  MoveL 3991 to (-40.74, 149.76, 69.25) mm, rotated rx -180 ry 0 rz 180 deg; joints [-126.379, -59.707, -80.826, 60.372, 67.852, -33.54]
  MoveL 3992 to (-40.74, 149.76, 69.25) mm, rotated rx -180 ry 0 rz 180 deg; joints [-126.379, -59.707, -80.826, 60.372, 67.852, -33.54]
  Call Extruder(12.04180)
  MoveL 3993 to (-40.78, 149.45, 69.25) mm, rotated rx 180 ry 0 rz 180 deg; joints [-126.398, -59.688, -80.879, 60.344, 67.858, -33.503]
  MoveL 3994 to (-40.78, 149.45, 69.25) mm, rotated rx 180 ry 0 rz 180 deg; joints [-126.398, -59.688, -80.879, 60.344, 67.858, -33.503]
  Call Extruder(12.20062)
  MoveL 3995 to (-40.83, 149.14, 69.25) mm, rotated rx 180 ry 0 rz -180 deg; joints [-126.417, -59.668, -80.931, 60.315, 67.863, -33.466]
  MoveL 3996 to (-40.83, 149.14, 69.25) mm, rotated rx 180 ry 0 rz -180 deg; joints [-126.417, -59.668, -80.931, 60.315, 67.863, -33.466]
  Call Extruder(12.37928)
  MoveL 3997 to (-40.88, 148.8, 69.25) mm, rotated rx 180 ry 0 rz 180 deg; joints [-126.439, -59.646, -80.989, 60.282, 67.869, -33.424]
  MoveL 3998 to (-40.88, 148.8, 69.25) mm, rotated rx 180 ry 0 rz 180 deg; joints [-126.439, -59.646, -80.989, 60.282, 67.869, -33.424]
  Call Extruder(12.57772)
  MoveL 3999 to (-40.92, 148.41, 69.25) mm, rotated rx 180 ry 0 rz 180 deg; joints [-126.465, -59.622, -81.054, 60.244, 67.875, -33.377]
  MoveL 4000 to (-40.92, 148.41, 69.25) mm, rotated rx 180 ry 0 rz 180 deg; joints [-126.465, -59.622, -81.054, 60.244, 67.875, -33.377]
  Call Extruder(12.77530)
  MoveL 4001 to (-40.97, 148.02, 69.25) mm, rotated rx 180 ry 0 rz 180 deg; joints [-126.491, -59.598, -81.118, 60.206, 67.881, -33.33]
  MoveL 4002 to (-40.97, 148.02, 69.25) mm, rotated rx 180 ry 0 rz 180 deg; joints [-126.491, -59.598, -81.118, 60.206, 67.881, -33.33]
  Call Extruder(12.97200)
  MoveL 4003 to (-41.02, 147.63, 69.25) mm, rotated rx 180 ry 0 rz 180 deg; joints [-126.517, -59.574, -81.183, 60.168, 67.886, -33.284]
  MoveL 4004 to (-41.02, 147.63, 69.25) mm, rotated rx 180 ry 0 rz 180 deg; joints [-126.517, -59.574, -81.183, 60.168, 67.886, -33.284]
  Call Extruder(13.16784)
  MoveL 4005 to (-41.06, 147.25, 69.25) mm, rotated rx 180 ry 0 rz 180 deg; joints [-126.543, -59.55, -81.247, 60.131, 67.892, -33.237]
  MoveL 4006 to (-41.06, 147.25, 69.25) mm, rotated rx 180 ry 0 rz 180 deg; joints [-126.543, -59.55, -81.247, 60.131, 67.892, -33.237]
  Call Extruder(13.46324)
  MoveL 4007 to (-41.11, 146.66, 69.25) mm, rotated rx 180 ry 0 rz 180 deg; joints [-126.585, -59.515, -81.342, 60.071, 67.899, -33.167]
  MoveL 4008 to (-41.11, 146.66, 69.25) mm, rotated rx 180 ry 0 rz 180 deg; joints [-126.585, -59.515, -81.342, 60.071, 67.899, -33.167]
  Call Extruder(13.75731)
  MoveL 4009 to (-41.15, 146.07, 69.25) mm, rotated rx -180 ry 0 rz 180 deg; joints [-126.628, -59.48, -81.437, 60.012, 67.906, -33.096]
  MoveL 4010 to (-41.15, 146.07, 69.25) mm, rotated rx -180 ry 0 rz 180 deg; joints [-126.628, -59.48, -81.437, 60.012, 67.906, -33.096]
  Call Extruder(14.05004)
  MoveL 4011 to (-41.2, 145.48, 69.25) mm, rotated rx -180 ry 0 rz -180 deg; joints [-126.67, -59.444, -81.532, 59.953, 67.912, -33.026]
  MoveL 4012 to (-41.2, 145.48, 69.25) mm, rotated rx -180 ry 0 rz -180 deg; joints [-126.67, -59.444, -81.532, 59.953, 67.912, -33.026]
  Call Extruder(14.62350)
  MoveL 4013 to (-41.25, 144.32, 69.25) mm, rotated rx 180 ry 0 rz -180 deg; joints [-126.759, -59.377, -81.714, 59.832, 67.921, -32.889]
  MoveL 4014 to (-41.25, 144.32, 69.25) mm, rotated rx 180 ry 0 rz -180 deg; joints [-126.759, -59.377, -81.714, 59.832, 67.921, -32.889]
  Call Extruder(15.33745)
  MoveL 4015 to (-41.29, 142.86, 69.25) mm, rotated rx 180 ry 0 rz 180 deg; joints [-126.873, -59.294, -81.938, 59.679, 67.931, -32.718]
  Call Extruder(57.40228)
  MoveL 4016 to (-41.29, 57.14, 69.25) mm, rotated rx 180 ry 0 rz 180 deg; joints [-135.148, -55.35, -93.55, 49.281, 68.519, -23.047]
  Call Extruder(57.83083)
  MoveL 4017 to (-41.27, 56.26, 69.25) mm, rotated rx -180 ry 0 rz 180 deg; joints [-135.25, -55.319, -93.653, 49.16, 68.526, -22.952]
  MoveL 4018 to (-41.27, 56.26, 69.25) mm, rotated rx -180 ry 0 rz 180 deg; joints [-135.25, -55.319, -93.653, 49.16, 68.526, -22.952]
  Call Extruder(58.40429)
  MoveL 4019 to (-41.23, 55.1, 69.25) mm, rotated rx -180 ry 0 rz -180 deg; joints [-135.387, -55.278, -93.786, 48.995, 68.534, -22.827]
  MoveL 4020 to (-41.23, 55.1, 69.25) mm, rotated rx -180 ry 0 rz -180 deg; joints [-135.387, -55.278, -93.786, 48.995, 68.534, -22.827]
  Call Extruder(58.83860)
  MoveL 4021 to (-41.18, 54.23, 69.25) mm, rotated rx 180 ry 0 rz 180 deg; joints [-135.493, -55.248, -93.885, 48.87, 68.538, -22.733]
  MoveL 4022 to (-41.18, 54.23, 69.25) mm, rotated rx 180 ry 0 rz 180 deg; joints [-135.493, -55.248, -93.885, 48.87, 68.538, -22.733]
  Call Extruder(59.13267)
  MoveL 4023 to (-41.13, 53.64, 69.25) mm, rotated rx -180 ry 0 rz 180 deg; joints [-135.566, -55.228, -93.95, 48.784, 68.539, -22.67]
  MoveL 4024 to (-41.13, 53.64, 69.25) mm, rotated rx -180 ry 0 rz 180 deg; joints [-135.566, -55.228, -93.95, 48.784, 68.539, -22.67]
  Call Extruder(59.42806)
  MoveL 4025 to (-41.09, 53.05, 69.25) mm, rotated rx -180 ry 0 rz 180 deg; joints [-135.64, -55.209, -94.014, 48.699, 68.541, -22.607]
  MoveL 4026 to (-41.09, 53.05, 69.25) mm, rotated rx -180 ry 0 rz 180 deg; joints [-135.64, -55.209, -94.014, 48.699, 68.541, -22.607]
  Call Extruder(59.67430)
  MoveL 4027 to (-41.04, 52.56, 69.25) mm, rotated rx 180 ry 0 rz -180 deg; joints [-135.701, -55.193, -94.066, 48.627, 68.541, -22.556]
  MoveL 4028 to (-41.04, 52.56, 69.25) mm, rotated rx 180 ry 0 rz -180 deg; joints [-135.701, -55.193, -94.066, 48.627, 68.541, -22.556]
  Call Extruder(59.87100)
  MoveL 4029 to (-40.99, 52.17, 69.25) mm, rotated rx -180 ry 0 rz 180 deg; joints [-135.751, -55.181, -94.107, 48.569, 68.54, -22.515]
  MoveL 4030 to (-40.99, 52.17, 69.25) mm, rotated rx -180 ry 0 rz 180 deg; joints [-135.751, -55.181, -94.107, 48.569, 68.54, -22.515]
  Call Extruder(60.06858)
  MoveL 4031 to (-40.95, 51.78, 69.25) mm, rotated rx 180 ry 0 rz -180 deg; joints [-135.801, -55.169, -94.147, 48.511, 68.54, -22.474]
  MoveL 4032 to (-40.95, 51.78, 69.25) mm, rotated rx 180 ry 0 rz -180 deg; joints [-135.801, -55.169, -94.147, 48.511, 68.54, -22.474]
  Call Extruder(60.26702)
  MoveL 4033 to (-40.9, 51.4, 69.25) mm, rotated rx 180 ry 0 rz -180 deg; joints [-135.852, -55.157, -94.187, 48.453, 68.539, -22.433]
  MoveL 4034 to (-40.9, 51.4, 69.25) mm, rotated rx 180 ry 0 rz -180 deg; joints [-135.852, -55.157, -94.187, 48.453, 68.539, -22.433]
  Call Extruder(60.46633)
  MoveL 4035 to (-40.86, 51.01, 69.25) mm, rotated rx 180 ry 0 rz 180 deg; joints [-135.902, -55.145, -94.227, 48.394, 68.539, -22.392]
  MoveL 4036 to (-40.86, 51.01, 69.25) mm, rotated rx 180 ry 0 rz 180 deg; joints [-135.902, -55.145, -94.227, 48.394, 68.539, -22.392]
  Call Extruder(60.62514)
  MoveL 4037 to (-40.81, 50.7, 69.25) mm, rotated rx 180 ry 0 rz -180 deg; joints [-135.943, -55.136, -94.257, 48.347, 68.537, -22.36]
  MoveL 4038 to (-40.81, 50.7, 69.25) mm, rotated rx 180 ry 0 rz -180 deg; joints [-135.943, -55.136, -94.257, 48.347, 68.537, -22.36]
  Call Extruder(60.78469)
  MoveL 4039 to (-40.76, 50.4, 69.25) mm, rotated rx 180 ry 0 rz -180 deg; joints [-135.984, -55.127, -94.287, 48.3, 68.535, -22.329]
  MoveL 4040 to (-40.76, 50.4, 69.25) mm, rotated rx 180 ry 0 rz -180 deg; joints [-135.984, -55.127, -94.287, 48.3, 68.535, -22.329]
  Call Extruder(60.94496)
  MoveL 4041 to (-40.71, 50.09, 69.25) mm, rotated rx 180 ry 0 rz 180 deg; joints [-136.025, -55.118, -94.317, 48.253, 68.534, -22.297]
  MoveL 4042 to (-40.71, 50.09, 69.25) mm, rotated rx 180 ry 0 rz 180 deg; joints [-136.025, -55.118, -94.317, 48.253, 68.534, -22.297]
  Call Extruder(61.10596)
  MoveL 4043 to (-40.66, 49.79, 69.25) mm, rotated rx 180 ry 0 rz -180 deg; joints [-136.067, -55.109, -94.347, 48.206, 68.532, -22.265]
  MoveL 4044 to (-40.66, 49.79, 69.25) mm, rotated rx 180 ry 0 rz -180 deg; joints [-136.067, -55.109, -94.347, 48.206, 68.532, -22.265]
  Call Extruder(61.26769)
  MoveL 4045 to (-40.61, 49.48, 69.25) mm, rotated rx 180 ry 0 rz 180 deg; joints [-136.108, -55.1, -94.377, 48.159, 68.53, -22.233]
  MoveL 4046 to (-40.61, 49.48, 69.25) mm, rotated rx 180 ry 0 rz 180 deg; joints [-136.108, -55.1, -94.377, 48.159, 68.53, -22.233]
  Call Extruder(61.43014)
  MoveL 4047 to (-40.56, 49.18, 69.25) mm, rotated rx 180 ry 0 rz 180 deg; joints [-136.149, -55.091, -94.407, 48.112, 68.529, -22.201]
  MoveL 4048 to (-40.56, 49.18, 69.25) mm, rotated rx 180 ry 0 rz 180 deg; joints [-136.149, -55.091, -94.407, 48.112, 68.529, -22.201]
  Call Extruder(61.56407)
  MoveL 4049 to (-40.52, 48.93, 69.25) mm, rotated rx 180 ry 0 rz 180 deg; joints [-136.184, -55.084, -94.43, 48.072, 68.526, -22.176]
  MoveL 4050 to (-40.52, 48.93, 69.25) mm, rotated rx 180 ry 0 rz 180 deg; joints [-136.184, -55.084, -94.43, 48.072, 68.526, -22.176]
  Call Extruder(61.69860)
  MoveL 4051 to (-40.47, 48.68, 69.25) mm, rotated rx 180 ry 0 rz 180 deg; joints [-136.219, -55.077, -94.453, 48.033, 68.524, -22.15]
  MoveL 4052 to (-40.47, 48.68, 69.25) mm, rotated rx 180 ry 0 rz 180 deg; joints [-136.219, -55.077, -94.453, 48.033, 68.524, -22.15]
  Call Extruder(61.83375)
  MoveL 4053 to (-40.42, 48.43, 69.25) mm, rotated rx -180 ry 0 rz -180 deg; joints [-136.254, -55.07, -94.476, 47.993, 68.522, -22.124]
  MoveL 4054 to (-40.42, 48.43, 69.25) mm, rotated rx -180 ry 0 rz -180 deg; joints [-136.254, -55.07, -94.476, 47.993, 68.522, -22.124]
  Call Extruder(61.96950)
  MoveL 4055 to (-40.37, 48.18, 69.25) mm, rotated rx -180 ry 0 rz 180 deg; joints [-136.288, -55.063, -94.499, 47.954, 68.519, -22.099]
  MoveL 4056 to (-40.37, 48.18, 69.25) mm, rotated rx -180 ry 0 rz 180 deg; joints [-136.288, -55.063, -94.499, 47.954, 68.519, -22.099]
  Call Extruder(62.10587)
  MoveL 4057 to (-40.32, 47.93, 69.25) mm, rotated rx 180 ry 0 rz 180 deg; joints [-136.323, -55.056, -94.522, 47.915, 68.517, -22.073]
  MoveL 4058 to (-40.32, 47.93, 69.25) mm, rotated rx 180 ry 0 rz 180 deg; joints [-136.323, -55.056, -94.522, 47.915, 68.517, -22.073]
  Call Extruder(62.24285)
  MoveL 4059 to (-40.27, 47.68, 69.25) mm, rotated rx -180 ry 0 rz 180 deg; joints [-136.358, -55.049, -94.545, 47.875, 68.515, -22.048]
  MoveL 4060 to (-40.27, 47.68, 69.25) mm, rotated rx -180 ry 0 rz 180 deg; joints [-136.358, -55.049, -94.545, 47.875, 68.515, -22.048]
  Call Extruder(62.38043)
  MoveL 4061 to (-40.22, 47.43, 69.25) mm, rotated rx 180 ry 0 rz 180 deg; joints [-136.393, -55.042, -94.568, 47.836, 68.512, -22.022]
  MoveL 4062 to (-40.22, 47.43, 69.25) mm, rotated rx 180 ry 0 rz 180 deg; joints [-136.393, -55.042, -94.568, 47.836, 68.512, -22.022]
  Call Extruder(62.49416)
  MoveL 4063 to (-40.17, 47.23, 69.25) mm, rotated rx -180 ry 0 rz -180 deg; joints [-136.422, -55.037, -94.587, 47.803, 68.51, -22.001]
  MoveL 4064 to (-40.17, 47.23, 69.25) mm, rotated rx -180 ry 0 rz -180 deg; joints [-136.422, -55.037, -94.587, 47.803, 68.51, -22.001]
  Call Extruder(62.60834)
  MoveL 4065 to (-40.13, 47.02, 69.25) mm, rotated rx 180 ry 0 rz 180 deg; joints [-136.452, -55.032, -94.605, 47.77, 68.508, -21.98]
  MoveL 4066 to (-40.13, 47.02, 69.25) mm, rotated rx 180 ry 0 rz 180 deg; joints [-136.452, -55.032, -94.605, 47.77, 68.508, -21.98]
  Call Extruder(62.72297)
  MoveL 4067 to (-40.08, 46.82, 69.25) mm, rotated rx 180 ry 0 rz 180 deg; joints [-136.481, -55.026, -94.623, 47.737, 68.506, -21.959]
  MoveL 4068 to (-40.08, 46.82, 69.25) mm, rotated rx 180 ry 0 rz 180 deg; joints [-136.481, -55.026, -94.623, 47.737, 68.506, -21.959]
  Call Extruder(62.83806)
  MoveL 4069 to (-40.04, 46.61, 69.25) mm, rotated rx 180 ry 0 rz 180 deg; joints [-136.51, -55.021, -94.641, 47.704, 68.503, -21.939]
  MoveL 4070 to (-40.04, 46.61, 69.25) mm, rotated rx 180 ry 0 rz 180 deg; joints [-136.51, -55.021, -94.641, 47.704, 68.503, -21.939]
  Call Extruder(62.96029)
  MoveL 4071 to (-39.98, 46.4, 69.25) mm, rotated rx 180 ry 0 rz 180 deg; joints [-136.542, -55.015, -94.659, 47.669, 68.5, -21.917]
  MoveL 4072 to (-39.98, 46.4, 69.25) mm, rotated rx 180 ry 0 rz 180 deg; joints [-136.542, -55.015, -94.659, 47.669, 68.5, -21.917]
  Call Extruder(63.08996)
  MoveL 4073 to (-39.92, 46.18, 69.25) mm, rotated rx 180 ry 0 rz -180 deg; joints [-136.576, -55.01, -94.677, 47.631, 68.496, -21.895]
  MoveL 4074 to (-39.92, 46.18, 69.25) mm, rotated rx 180 ry 0 rz -180 deg; joints [-136.576, -55.01, -94.677, 47.631, 68.496, -21.895]
  Call Extruder(63.22019)
  MoveL 4075 to (-39.85, 45.95, 69.25) mm, rotated rx 180 ry 0 rz 180 deg; joints [-136.61, -55.005, -94.695, 47.594, 68.491, -21.872]
  MoveL 4076 to (-39.85, 45.95, 69.25) mm, rotated rx 180 ry 0 rz 180 deg; joints [-136.61, -55.005, -94.695, 47.594, 68.491, -21.872]
  Call Extruder(63.35098)
  MoveL 4077 to (-39.78, 45.73, 69.25) mm, rotated rx 180 ry 0 rz 180 deg; joints [-136.644, -55, -94.712, 47.556, 68.487, -21.85]
  MoveL 4078 to (-39.78, 45.73, 69.25) mm, rotated rx 180 ry 0 rz 180 deg; joints [-136.644, -55, -94.712, 47.556, 68.487, -21.85]
  Call Extruder(63.48234)
  MoveL 4079 to (-39.71, 45.51, 69.25) mm, rotated rx 180 ry 0 rz 180 deg; joints [-136.678, -54.994, -94.73, 47.518, 68.483, -21.828]
  MoveL 4080 to (-39.71, 45.51, 69.25) mm, rotated rx 180 ry 0 rz 180 deg; joints [-136.678, -54.994, -94.73, 47.518, 68.483, -21.828]
  Call Extruder(63.59424)
  MoveL 4081 to (-39.65, 45.32, 69.25) mm, rotated rx 180 ry 0 rz -180 deg; joints [-136.707, -54.99, -94.744, 47.486, 68.478, -21.809]
  MoveL 4082 to (-39.65, 45.32, 69.25) mm, rotated rx 180 ry 0 rz -180 deg; joints [-136.707, -54.99, -94.744, 47.486, 68.478, -21.809]
  Call Extruder(63.70659)
  MoveL 4083 to (-39.59, 45.13, 69.25) mm, rotated rx 180 ry 0 rz 180 deg; joints [-136.737, -54.986, -94.758, 47.454, 68.474, -21.79]
  MoveL 4084 to (-39.59, 45.13, 69.25) mm, rotated rx 180 ry 0 rz 180 deg; joints [-136.737, -54.986, -94.758, 47.454, 68.474, -21.79]
  Call Extruder(63.81938)
  MoveL 4085 to (-39.53, 44.94, 69.25) mm, rotated rx -180 ry 0 rz 180 deg; joints [-136.766, -54.982, -94.773, 47.422, 68.47, -21.772]
  MoveL 4086 to (-39.53, 44.94, 69.25) mm, rotated rx -180 ry 0 rz 180 deg; joints [-136.766, -54.982, -94.773, 47.422, 68.47, -21.772]
  Call Extruder(63.93261)
  MoveL 4087 to (-39.47, 44.75, 69.25) mm, rotated rx 180 ry 0 rz -180 deg; joints [-136.796, -54.977, -94.787, 47.39, 68.466, -21.753]
  MoveL 4088 to (-39.47, 44.75, 69.25) mm, rotated rx 180 ry 0 rz -180 deg; joints [-136.796, -54.977, -94.787, 47.39, 68.466, -21.753]
  Call Extruder(64.04629)
  MoveL 4089 to (-39.41, 44.56, 69.25) mm, rotated rx -180 ry 0 rz 180 deg; joints [-136.825, -54.973, -94.801, 47.358, 68.462, -21.734]
  MoveL 4090 to (-39.41, 44.56, 69.25) mm, rotated rx -180 ry 0 rz 180 deg; joints [-136.825, -54.973, -94.801, 47.358, 68.462, -21.734]
  Call Extruder(64.22825)
  MoveL 4091 to (-39.29, 44.27, 69.25) mm, rotated rx -180 ry 0 rz -180 deg; joints [-136.873, -54.968, -94.82, 47.305, 68.453, -21.706]
  MoveL 4092 to (-39.29, 44.27, 69.25) mm, rotated rx -180 ry 0 rz -180 deg; joints [-136.873, -54.968, -94.82, 47.305, 68.453, -21.706]
  Call Extruder(64.41097)
  MoveL 4093 to (-39.16, 43.98, 69.25) mm, rotated rx 180 ry 0 rz -180 deg; joints [-136.922, -54.962, -94.839, 47.253, 68.444, -21.678]
  MoveL 4094 to (-39.16, 43.98, 69.25) mm, rotated rx 180 ry 0 rz -180 deg; joints [-136.922, -54.962, -94.839, 47.253, 68.444, -21.678]
  Call Extruder(64.58138)
  MoveL 4095 to (-39.05, 43.71, 69.25) mm, rotated rx 180 ry 0 rz 180 deg; joints [-136.967, -54.957, -94.856, 47.205, 68.436, -21.652]
  MoveL 4096 to (-39.05, 43.71, 69.25) mm, rotated rx 180 ry 0 rz 180 deg; joints [-136.967, -54.957, -94.856, 47.205, 68.436, -21.652]
  Call Extruder(64.73937)
  MoveL 4097 to (-38.94, 43.46, 69.25) mm, rotated rx 180 ry 0 rz -180 deg; joints [-137.009, -54.952, -94.871, 47.16, 68.427, -21.628]
  MoveL 4098 to (-38.94, 43.46, 69.25) mm, rotated rx 180 ry 0 rz -180 deg; joints [-137.009, -54.952, -94.871, 47.16, 68.427, -21.628]
  Call Extruder(64.89795)
  MoveL 4099 to (-38.84, 43.21, 69.25) mm, rotated rx 180 ry 0 rz 180 deg; joints [-137.05, -54.948, -94.886, 47.115, 68.419, -21.604]
  MoveL 4100 to (-38.84, 43.21, 69.25) mm, rotated rx 180 ry 0 rz 180 deg; joints [-137.05, -54.948, -94.886, 47.115, 68.419, -21.604]
  Call Extruder(65.10412)
  MoveL 4101 to (-38.66, 42.91, 69.25) mm, rotated rx 180 ry 0 rz -180 deg; joints [-137.107, -54.944, -94.9, 47.056, 68.405, -21.576]
  MoveL 4102 to (-38.66, 42.91, 69.25) mm, rotated rx 180 ry 0 rz -180 deg; joints [-137.107, -54.944, -94.9, 47.056, 68.405, -21.576]
  Call Extruder(65.31106)
  MoveL 4103 to (-38.49, 42.6, 69.25) mm, rotated rx 180 ry 0 rz 180 deg; joints [-137.163, -54.94, -94.913, 46.997, 68.391, -21.548]
  MoveL 4104 to (-38.49, 42.6, 69.25) mm, rotated rx 180 ry 0 rz 180 deg; joints [-137.163, -54.94, -94.913, 46.997, 68.391, -21.548]
  Call Extruder(65.51879)
  MoveL 4105 to (-38.31, 42.3, 69.25) mm, rotated rx 180 ry 0 rz 180 deg; joints [-137.219, -54.936, -94.926, 46.938, 68.377, -21.52]
  MoveL 4106 to (-38.31, 42.3, 69.25) mm, rotated rx 180 ry 0 rz 180 deg; joints [-137.219, -54.936, -94.926, 46.938, 68.377, -21.52]
  Call Extruder(65.72729)
  MoveL 4107 to (-38.13, 41.99, 69.25) mm, rotated rx 180 ry 0 rz 180 deg; joints [-137.275, -54.932, -94.939, 46.879, 68.362, -21.492]
  MoveL 4108 to (-38.13, 41.99, 69.25) mm, rotated rx 180 ry 0 rz 180 deg; joints [-137.275, -54.932, -94.939, 46.879, 68.362, -21.492]
  Call Extruder(65.90684)
  MoveL 4109 to (-37.96, 41.75, 69.25) mm, rotated rx 180 ry 0 rz 180 deg; joints [-137.324, -54.93, -94.945, 46.829, 68.347, -21.471]
  MoveL 4110 to (-37.96, 41.75, 69.25) mm, rotated rx 180 ry 0 rz 180 deg; joints [-137.324, -54.93, -94.945, 46.829, 68.347, -21.471]
  Call Extruder(66.24028)
  MoveL 4111 to (-37.63, 41.3, 69.25) mm, rotated rx 180 ry 0 rz 180 deg; joints [-137.415, -54.927, -94.956, 46.736, 68.319, -21.431]
  MoveL 4112 to (-37.63, 41.3, 69.25) mm, rotated rx 180 ry 0 rz 180 deg; joints [-137.415, -54.927, -94.956, 46.736, 68.319, -21.431]
  Call Extruder(66.57490)
  MoveL 4113 to (-37.3, 40.85, 69.25) mm, rotated rx 180 ry 0 rz 180 deg; joints [-137.506, -54.924, -94.967, 46.642, 68.291, -21.392]
  Call Extruder(67.40283)
  MoveL 4114 to (-36.39, 39.81, 69.25) mm, rotated rx 180 ry 0 rz -180 deg; joints [-137.733, -54.923, -94.971, 46.414, 68.211, -21.305]
  Call Extruder(68.23074)
  MoveL 4115 to (-35.35, 38.9, 69.25) mm, rotated rx 180 ry 0 rz -180 deg; joints [-137.958, -54.931, -94.945, 46.193, 68.116, -21.235]
  Call Extruder(68.39804)
  MoveL 4116 to (-35.13, 38.73, 69.25) mm, rotated rx -180 ry 0 rz 180 deg; joints [-138.003, -54.934, -94.935, 46.15, 68.095, -21.224]
  MoveL 4117 to (-35.13, 38.73, 69.25) mm, rotated rx -180 ry 0 rz 180 deg; joints [-138.003, -54.934, -94.935, 46.15, 68.095, -21.224]
  Call Extruder(68.73147)
  MoveL 4118 to (-34.68, 38.41, 69.25) mm, rotated rx 180 ry 0 rz 180 deg; joints [-138.092, -54.939, -94.915, 46.064, 68.053, -21.201]
  MoveL 4119 to (-34.68, 38.41, 69.25) mm, rotated rx 180 ry 0 rz 180 deg; joints [-138.092, -54.939, -94.915, 46.064, 68.053, -21.201]
  Call Extruder(69.06371)
  MoveL 4120 to (-34.22, 38.08, 69.25) mm, rotated rx 180 ry 0 rz -180 deg; joints [-138.182, -54.945, -94.896, 45.978, 68.011, -21.178]
  MoveL 4121 to (-34.22, 38.08, 69.25) mm, rotated rx 180 ry 0 rz -180 deg; joints [-138.182, -54.945, -94.896, 45.978, 68.011, -21.178]
  Call Extruder(69.18141)
  MoveL 4122 to (-34.05, 37.98, 69.25) mm, rotated rx 180 ry 0 rz 180 deg; joints [-138.213, -54.948, -94.885, 45.949, 67.995, -21.172]
  MoveL 4123 to (-34.05, 37.98, 69.25) mm, rotated rx 180 ry 0 rz 180 deg; joints [-138.213, -54.948, -94.885, 45.949, 67.995, -21.172]
  Call Extruder(69.38913)
  MoveL 4124 to (-33.75, 37.8, 69.25) mm, rotated rx -180 ry 0 rz -180 deg; joints [-138.267, -54.954, -94.867, 45.898, 67.966, -21.162]
  MoveL 4125 to (-33.75, 37.8, 69.25) mm, rotated rx -180 ry 0 rz -180 deg; joints [-138.267, -54.954, -94.867, 45.898, 67.966, -21.162]
  Call Extruder(69.59607)
  MoveL 4126 to (-33.45, 37.63, 69.25) mm, rotated rx 180 ry 0 rz 180 deg; joints [-138.322, -54.959, -94.848, 45.847, 67.937, -21.151]
  MoveL 4127 to (-33.45, 37.63, 69.25) mm, rotated rx 180 ry 0 rz 180 deg; joints [-138.322, -54.959, -94.848, 45.847, 67.937, -21.151]
  Call Extruder(69.80224)
  MoveL 4128 to (-33.14, 37.45, 69.25) mm, rotated rx -180 ry 0 rz 180 deg; joints [-138.376, -54.965, -94.83, 45.796, 67.909, -21.141]
  MoveL 4129 to (-33.14, 37.45, 69.25) mm, rotated rx -180 ry 0 rz 180 deg; joints [-138.376, -54.965, -94.83, 45.796, 67.909, -21.141]
  Call Extruder(69.98392)
  MoveL 4130 to (-32.87, 37.31, 69.25) mm, rotated rx 180 ry 0 rz 180 deg; joints [-138.424, -54.97, -94.811, 45.752, 67.882, -21.133]
  MoveL 4131 to (-32.87, 37.31, 69.25) mm, rotated rx 180 ry 0 rz 180 deg; joints [-138.424, -54.97, -94.811, 45.752, 67.882, -21.133]
  Call Extruder(70.14192)
  MoveL 4132 to (-32.62, 37.2, 69.25) mm, rotated rx 180 ry 0 rz -180 deg; joints [-138.464, -54.976, -94.791, 45.716, 67.858, -21.128]
  MoveL 4133 to (-32.62, 37.2, 69.25) mm, rotated rx 180 ry 0 rz -180 deg; joints [-138.464, -54.976, -94.791, 45.716, 67.858, -21.128]
  Call Extruder(70.29931)
  MoveL 4134 to (-32.37, 37.1, 69.25) mm, rotated rx 180 ry 0 rz 180 deg; joints [-138.504, -54.982, -94.772, 45.679, 67.834, -21.124]
  MoveL 4135 to (-32.37, 37.1, 69.25) mm, rotated rx 180 ry 0 rz 180 deg; joints [-138.504, -54.982, -94.772, 45.679, 67.834, -21.124]
  Call Extruder(70.48203)
  MoveL 4136 to (-32.07, 36.98, 69.25) mm, rotated rx 180 ry 0 rz 180 deg; joints [-138.551, -54.989, -94.748, 45.637, 67.806, -21.119]
  MoveL 4137 to (-32.07, 36.98, 69.25) mm, rotated rx 180 ry 0 rz 180 deg; joints [-138.551, -54.989, -94.748, 45.637, 67.806, -21.119]
  Call Extruder(70.66398)
  MoveL 4138 to (-31.78, 36.85, 69.25) mm, rotated rx -180 ry 0 rz 180 deg; joints [-138.597, -54.996, -94.725, 45.595, 67.778, -21.114]
  MoveL 4139 to (-31.78, 36.85, 69.25) mm, rotated rx -180 ry 0 rz 180 deg; joints [-138.597, -54.996, -94.725, 45.595, 67.778, -21.114]
  Call Extruder(70.81131)
  MoveL 4140 to (-31.54, 36.76, 69.25) mm, rotated rx 180 ry 0 rz 180 deg; joints [-138.634, -55.002, -94.705, 45.562, 67.754, -21.111]
  MoveL 4141 to (-31.54, 36.76, 69.25) mm, rotated rx 180 ry 0 rz 180 deg; joints [-138.634, -55.002, -94.705, 45.562, 67.754, -21.111]
  Call Extruder(70.92455)
  MoveL 4142 to (-31.35, 36.7, 69.25) mm, rotated rx 180 ry 0 rz 180 deg; joints [-138.662, -55.007, -94.688, 45.537, 67.736, -21.109]
  MoveL 4143 to (-31.35, 36.7, 69.25) mm, rotated rx 180 ry 0 rz 180 deg; joints [-138.662, -55.007, -94.688, 45.537, 67.736, -21.109]
  Call Extruder(71.03734)
  MoveL 4144 to (-31.17, 36.64, 69.25) mm, rotated rx 180 ry 0 rz 180 deg; joints [-138.69, -55.012, -94.67, 45.513, 67.718, -21.108]
  MoveL 4145 to (-31.17, 36.64, 69.25) mm, rotated rx 180 ry 0 rz 180 deg; joints [-138.69, -55.012, -94.67, 45.513, 67.718, -21.108]
  Call Extruder(71.14968)
  MoveL 4146 to (-30.98, 36.58, 69.25) mm, rotated rx -180 ry 0 rz 180 deg; joints [-138.718, -55.017, -94.653, 45.488, 67.699, -21.106]
  MoveL 4147 to (-30.98, 36.58, 69.25) mm, rotated rx -180 ry 0 rz 180 deg; joints [-138.718, -55.017, -94.653, 45.488, 67.699, -21.106]
  Call Extruder(71.26159)
  MoveL 4148 to (-30.79, 36.52, 69.25) mm, rotated rx 180 ry 0 rz 180 deg; joints [-138.745, -55.022, -94.636, 45.464, 67.681, -21.105]
  MoveL 4149 to (-30.79, 36.52, 69.25) mm, rotated rx 180 ry 0 rz 180 deg; joints [-138.745, -55.022, -94.636, 45.464, 67.681, -21.105]
  Call Extruder(71.38299)
  MoveL 4150 to (-30.58, 36.45, 69.25) mm, rotated rx -180 ry 0 rz 180 deg; joints [-138.776, -55.028, -94.617, 45.437, 67.661, -21.104]
  MoveL 4151 to (-30.58, 36.45, 69.25) mm, rotated rx -180 ry 0 rz 180 deg; joints [-138.776, -55.028, -94.617, 45.437, 67.661, -21.104]
  Call Extruder(71.51378)
  MoveL 4152 to (-30.36, 36.39, 69.25) mm, rotated rx -180 ry 0 rz 180 deg; joints [-138.808, -55.034, -94.597, 45.409, 67.639, -21.102]
  MoveL 4153 to (-30.36, 36.39, 69.25) mm, rotated rx -180 ry 0 rz 180 deg; joints [-138.808, -55.034, -94.597, 45.409, 67.639, -21.102]
  Call Extruder(71.64400)
  MoveL 4154 to (-30.14, 36.32, 69.25) mm, rotated rx 180 ry 0 rz 180 deg; joints [-138.84, -55.04, -94.576, 45.381, 67.617, -21.101]
  MoveL 4155 to (-30.14, 36.32, 69.25) mm, rotated rx 180 ry 0 rz 180 deg; joints [-138.84, -55.04, -94.576, 45.381, 67.617, -21.101]
  Call Extruder(71.77367)
  MoveL 4156 to (-29.91, 36.25, 69.25) mm, rotated rx 180 ry 0 rz -180 deg; joints [-138.873, -55.046, -94.555, 45.352, 67.595, -21.1]
  MoveL 4157 to (-29.91, 36.25, 69.25) mm, rotated rx 180 ry 0 rz -180 deg; joints [-138.873, -55.046, -94.555, 45.352, 67.595, -21.1]
  Call Extruder(71.90276)
  MoveL 4158 to (-29.69, 36.18, 69.25) mm, rotated rx 180 ry 0 rz -180 deg; joints [-138.905, -55.053, -94.534, 45.324, 67.573, -21.099]
  MoveL 4159 to (-29.69, 36.18, 69.25) mm, rotated rx 180 ry 0 rz -180 deg; joints [-138.905, -55.053, -94.534, 45.324, 67.573, -21.099]
  Call Extruder(72.01784)
  MoveL 4160 to (-29.48, 36.14, 69.25) mm, rotated rx 180 ry 0 rz 180 deg; joints [-138.932, -55.059, -94.513, 45.301, 67.553, -21.1]
  MoveL 4161 to (-29.48, 36.14, 69.25) mm, rotated rx 180 ry 0 rz 180 deg; joints [-138.932, -55.059, -94.513, 45.301, 67.553, -21.1]
  Call Extruder(72.13246)
  MoveL 4162 to (-29.28, 36.09, 69.25) mm, rotated rx -180 ry 0 rz -180 deg; joints [-138.96, -55.065, -94.492, 45.278, 67.532, -21.101]
  MoveL 4163 to (-29.28, 36.09, 69.25) mm, rotated rx -180 ry 0 rz -180 deg; joints [-138.96, -55.065, -94.492, 45.278, 67.532, -21.101]
  Call Extruder(72.24663)
  MoveL 4164 to (-29.08, 36.05, 69.25) mm, rotated rx 180 ry 0 rz -180 deg; joints [-138.987, -55.072, -94.471, 45.254, 67.512, -21.102]
  MoveL 4165 to (-29.08, 36.05, 69.25) mm, rotated rx 180 ry 0 rz -180 deg; joints [-138.987, -55.072, -94.471, 45.254, 67.512, -21.102]
  Call Extruder(72.36034)
  MoveL 4166 to (-28.87, 36, 69.25) mm, rotated rx -180 ry 0 rz -180 deg; joints [-139.014, -55.078, -94.449, 45.231, 67.492, -21.102]
  MoveL 4167 to (-28.87, 36, 69.25) mm, rotated rx -180 ry 0 rz -180 deg; joints [-139.014, -55.078, -94.449, 45.231, 67.492, -21.102]
  Call Extruder(72.48576)
  MoveL 4168 to (-28.64, 35.96, 69.25) mm, rotated rx 180 ry 0 rz 180 deg; joints [-139.044, -55.085, -94.426, 45.206, 67.469, -21.104]
  MoveL 4169 to (-28.64, 35.96, 69.25) mm, rotated rx 180 ry 0 rz 180 deg; joints [-139.044, -55.085, -94.426, 45.206, 67.469, -21.104]
  Call Extruder(72.62274)
  MoveL 4170 to (-28.4, 35.91, 69.25) mm, rotated rx -180 ry 0 rz -180 deg; joints [-139.077, -55.093, -94.4, 45.178, 67.445, -21.105]
  MoveL 4171 to (-28.4, 35.91, 69.25) mm, rotated rx -180 ry 0 rz -180 deg; joints [-139.077, -55.093, -94.4, 45.178, 67.445, -21.105]
  Call Extruder(72.75911)
  MoveL 4172 to (-28.15, 35.86, 69.25) mm, rotated rx 180 ry 0 rz 180 deg; joints [-139.109, -55.101, -94.373, 45.151, 67.42, -21.107]
  MoveL 4173 to (-28.15, 35.86, 69.25) mm, rotated rx 180 ry 0 rz 180 deg; joints [-139.109, -55.101, -94.373, 45.151, 67.42, -21.107]
  Call Extruder(72.89487)
  MoveL 4174 to (-27.9, 35.81, 69.25) mm, rotated rx 180 ry 0 rz 180 deg; joints [-139.142, -55.109, -94.347, 45.123, 67.395, -21.108]
  MoveL 4175 to (-27.9, 35.81, 69.25) mm, rotated rx 180 ry 0 rz 180 deg; joints [-139.142, -55.109, -94.347, 45.123, 67.395, -21.108]
  Call Extruder(73.03001)
  MoveL 4176 to (-27.65, 35.76, 69.25) mm, rotated rx -180 ry 0 rz 180 deg; joints [-139.174, -55.117, -94.32, 45.096, 67.37, -21.11]
  MoveL 4177 to (-27.65, 35.76, 69.25) mm, rotated rx -180 ry 0 rz 180 deg; joints [-139.174, -55.117, -94.32, 45.096, 67.37, -21.11]
  Call Extruder(73.16455)
  MoveL 4178 to (-27.4, 35.71, 69.25) mm, rotated rx 180 ry 0 rz -180 deg; joints [-139.207, -55.125, -94.294, 45.068, 67.346, -21.111]
  MoveL 4179 to (-27.4, 35.71, 69.25) mm, rotated rx 180 ry 0 rz -180 deg; joints [-139.207, -55.125, -94.294, 45.068, 67.346, -21.111]
  Call Extruder(73.29848)
  MoveL 4180 to (-27.15, 35.66, 69.25) mm, rotated rx 180 ry 0 rz 180 deg; joints [-139.239, -55.133, -94.267, 45.041, 67.321, -21.113]
  MoveL 4181 to (-27.15, 35.66, 69.25) mm, rotated rx 180 ry 0 rz 180 deg; joints [-139.239, -55.133, -94.267, 45.041, 67.321, -21.113]
  Call Extruder(73.44634)
  MoveL 4182 to (-26.87, 35.61, 69.25) mm, rotated rx 180 ry 0 rz -180 deg; joints [-139.275, -55.142, -94.237, 45.012, 67.293, -21.115]
  MoveL 4183 to (-26.87, 35.61, 69.25) mm, rotated rx 180 ry 0 rz -180 deg; joints [-139.275, -55.142, -94.237, 45.012, 67.293, -21.115]
  Call Extruder(73.60807)
  MoveL 4184 to (-26.57, 35.56, 69.25) mm, rotated rx 180 ry 0 rz 180 deg; joints [-139.313, -55.152, -94.203, 44.98, 67.263, -21.118]
  MoveL 4185 to (-26.57, 35.56, 69.25) mm, rotated rx 180 ry 0 rz 180 deg; joints [-139.313, -55.152, -94.203, 44.98, 67.263, -21.118]
  Call Extruder(73.76908)
  MoveL 4186 to (-26.26, 35.51, 69.25) mm, rotated rx 180 ry 0 rz 180 deg; joints [-139.351, -55.162, -94.169, 44.948, 67.232, -21.122]
  MoveL 4187 to (-26.26, 35.51, 69.25) mm, rotated rx 180 ry 0 rz 180 deg; joints [-139.351, -55.162, -94.169, 44.948, 67.232, -21.122]
  Call Extruder(73.92935)
  MoveL 4188 to (-25.96, 35.47, 69.25) mm, rotated rx 180 ry 0 rz -180 deg; joints [-139.39, -55.172, -94.136, 44.917, 67.202, -21.125]
  MoveL 4189 to (-25.96, 35.47, 69.25) mm, rotated rx 180 ry 0 rz -180 deg; joints [-139.39, -55.172, -94.136, 44.917, 67.202, -21.125]
  Call Extruder(74.08890)
  MoveL 4190 to (-25.65, 35.42, 69.25) mm, rotated rx 180 ry 0 rz -180 deg; joints [-139.428, -55.182, -94.102, 44.885, 67.171, -21.128]
  MoveL 4191 to (-25.65, 35.42, 69.25) mm, rotated rx 180 ry 0 rz -180 deg; joints [-139.428, -55.182, -94.102, 44.885, 67.171, -21.128]
  Call Extruder(74.24773)
  MoveL 4192 to (-25.34, 35.37, 69.25) mm, rotated rx 180 ry 0 rz 180 deg; joints [-139.466, -55.193, -94.068, 44.853, 67.14, -21.131]
  MoveL 4193 to (-25.34, 35.37, 69.25) mm, rotated rx 180 ry 0 rz 180 deg; joints [-139.466, -55.193, -94.068, 44.853, 67.14, -21.131]
  Call Extruder(74.42640)
  MoveL 4194 to (-25, 35.32, 69.25) mm, rotated rx 180 ry 0 rz -180 deg; joints [-139.508, -55.205, -94.028, 44.819, 67.106, -21.136]
  MoveL 4195 to (-25, 35.32, 69.25) mm, rotated rx 180 ry 0 rz -180 deg; joints [-139.508, -55.205, -94.028, 44.819, 67.106, -21.136]
  Call Extruder(74.62484)
  MoveL 4196 to (-24.61, 35.27, 69.25) mm, rotated rx -180 ry 0 rz 180 deg; joints [-139.554, -55.218, -93.983, 44.781, 67.067, -21.141]
  MoveL 4197 to (-24.61, 35.27, 69.25) mm, rotated rx -180 ry 0 rz 180 deg; joints [-139.554, -55.218, -93.983, 44.781, 67.067, -21.141]
  Call Extruder(74.82241)
  MoveL 4198 to (-24.22, 35.23, 69.25) mm, rotated rx -180 ry 0 rz -180 deg; joints [-139.6, -55.232, -93.938, 44.744, 67.028, -21.147]
  MoveL 4199 to (-24.22, 35.23, 69.25) mm, rotated rx -180 ry 0 rz -180 deg; joints [-139.6, -55.232, -93.938, 44.744, 67.028, -21.147]
  Call Extruder(75.01912)
  MoveL 4200 to (-23.83, 35.18, 69.25) mm, rotated rx 180 ry 0 rz 180 deg; joints [-139.647, -55.246, -93.893, 44.707, 66.989, -21.153]
  MoveL 4201 to (-23.83, 35.18, 69.25) mm, rotated rx 180 ry 0 rz 180 deg; joints [-139.647, -55.246, -93.893, 44.707, 66.989, -21.153]
  Call Extruder(75.21496)
  MoveL 4202 to (-23.45, 35.14, 69.25) mm, rotated rx 180 ry 0 rz 180 deg; joints [-139.693, -55.259, -93.848, 44.669, 66.95, -21.159]
  MoveL 4203 to (-23.45, 35.14, 69.25) mm, rotated rx 180 ry 0 rz 180 deg; joints [-139.693, -55.259, -93.848, 44.669, 66.95, -21.159]
  Call Extruder(75.51035)
  MoveL 4204 to (-22.86, 35.09, 69.25) mm, rotated rx 180 ry 0 rz 180 deg; joints [-139.76, -55.281, -93.777, 44.616, 66.89, -21.17]
  MoveL 4205 to (-22.86, 35.09, 69.25) mm, rotated rx 180 ry 0 rz 180 deg; joints [-139.76, -55.281, -93.777, 44.616, 66.89, -21.17]
  Call Extruder(75.80442)
  MoveL 4206 to (-22.27, 35.05, 69.25) mm, rotated rx 180 ry 0 rz 180 deg; joints [-139.826, -55.303, -93.705, 44.563, 66.831, -21.181]
  MoveL 4207 to (-22.27, 35.05, 69.25) mm, rotated rx 180 ry 0 rz 180 deg; joints [-139.826, -55.303, -93.705, 44.563, 66.831, -21.181]
  Call Extruder(76.09715)
  MoveL 4208 to (-21.68, 35, 69.25) mm, rotated rx 180 ry 0 rz -180 deg; joints [-139.893, -55.324, -93.634, 44.511, 66.771, -21.192]
  MoveL 4209 to (-21.68, 35, 69.25) mm, rotated rx 180 ry 0 rz -180 deg; joints [-139.893, -55.324, -93.634, 44.511, 66.771, -21.192]
  Call Extruder(76.67060)
  MoveL 4210 to (-20.52, 34.95, 69.25) mm, rotated rx -180 ry 0 rz -180 deg; joints [-140.019, -55.369, -93.487, 44.414, 66.653, -21.22]
  MoveL 4211 to (-20.52, 34.95, 69.25) mm, rotated rx -180 ry 0 rz -180 deg; joints [-140.019, -55.369, -93.487, 44.414, 66.653, -21.22]
  Call Extruder(77.38456)
  MoveL 4212 to (-19.06, 34.91, 69.25) mm, rotated rx 180 ry 0 rz -180 deg; joints [-140.173, -55.426, -93.301, 44.296, 66.505, -21.256]
  Call Extruder(194.23128)
  MoveL 4213 to (219.06, 34.91, 69.25) mm, rotated rx 180 ry 0 rz 180 deg; joints [-155.896, -72.312, -50.804, 39.314, 40.134, -32.05]
  Call Extruder(194.65984)
  MoveL 4214 to (219.94, 34.93, 69.25) mm, rotated rx 180 ry 0 rz 180 deg; joints [-155.931, -72.411, -50.586, 39.358, 40.024, -32.132]
  MoveL 4215 to (219.94, 34.93, 69.25) mm, rotated rx 180 ry 0 rz 180 deg; joints [-155.931, -72.411, -50.586, 39.358, 40.024, -32.132]
  Call Extruder(195.23329)
  MoveL 4216 to (221.1, 34.97, 69.25) mm, rotated rx 180 ry 0 rz 180 deg; joints [-155.975, -72.545, -50.293, 39.421, 39.877, -32.245]
  MoveL 4217 to (221.1, 34.97, 69.25) mm, rotated rx 180 ry 0 rz 180 deg; joints [-155.975, -72.545, -50.293, 39.421, 39.877, -32.245]
  Call Extruder(195.66760)
  MoveL 4218 to (221.97, 35.02, 69.25) mm, rotated rx 180 ry 0 rz 180 deg; joints [-156.007, -72.647, -50.07, 39.471, 39.767, -32.333]
  MoveL 4219 to (221.97, 35.02, 69.25) mm, rotated rx 180 ry 0 rz 180 deg; joints [-156.007, -72.647, -50.07, 39.471, 39.767, -32.333]
  Call Extruder(195.96166)
  MoveL 4220 to (222.56, 35.07, 69.25) mm, rotated rx 180 ry 0 rz 180 deg; joints [-156.027, -72.716, -49.918, 39.508, 39.692, -32.396]
  MoveL 4221 to (222.56, 35.07, 69.25) mm, rotated rx 180 ry 0 rz 180 deg; joints [-156.027, -72.716, -49.918, 39.508, 39.692, -32.396]
  Call Extruder(196.25705)
  MoveL 4222 to (223.15, 35.11, 69.25) mm, rotated rx 180 ry 0 rz -180 deg; joints [-156.047, -72.786, -49.765, 39.546, 39.617, -32.458]
  MoveL 4223 to (223.15, 35.11, 69.25) mm, rotated rx 180 ry 0 rz -180 deg; joints [-156.047, -72.786, -49.765, 39.546, 39.617, -32.458]
  Call Extruder(196.50328)
  MoveL 4224 to (223.64, 35.16, 69.25) mm, rotated rx 180 ry 0 rz 180 deg; joints [-156.062, -72.844, -49.637, 39.578, 39.555, -32.511]
  MoveL 4225 to (223.64, 35.16, 69.25) mm, rotated rx 180 ry 0 rz 180 deg; joints [-156.062, -72.844, -49.637, 39.578, 39.555, -32.511]
  Call Extruder(196.69999)
  MoveL 4226 to (224.03, 35.21, 69.25) mm, rotated rx 180 ry 0 rz 180 deg; joints [-156.074, -72.891, -49.535, 39.606, 39.506, -32.555]
  MoveL 4227 to (224.03, 35.21, 69.25) mm, rotated rx 180 ry 0 rz 180 deg; joints [-156.074, -72.891, -49.535, 39.606, 39.506, -32.555]
  Call Extruder(196.89757)
  MoveL 4228 to (224.42, 35.25, 69.25) mm, rotated rx -180 ry 0 rz 180 deg; joints [-156.086, -72.938, -49.432, 39.634, 39.457, -32.599]
  MoveL 4229 to (224.42, 35.25, 69.25) mm, rotated rx -180 ry 0 rz 180 deg; joints [-156.086, -72.938, -49.432, 39.634, 39.457, -32.599]
  Call Extruder(197.09601)
  MoveL 4230 to (224.8, 35.3, 69.25) mm, rotated rx 180 ry 0 rz 180 deg; joints [-156.097, -72.985, -49.329, 39.662, 39.408, -32.643]
  MoveL 4231 to (224.8, 35.3, 69.25) mm, rotated rx 180 ry 0 rz 180 deg; joints [-156.097, -72.985, -49.329, 39.662, 39.408, -32.643]
  Call Extruder(197.29532)
  MoveL 4232 to (225.19, 35.34, 69.25) mm, rotated rx 180 ry 0 rz 180 deg; joints [-156.109, -73.032, -49.226, 39.69, 39.358, -32.688]
  MoveL 4233 to (225.19, 35.34, 69.25) mm, rotated rx 180 ry 0 rz 180 deg; joints [-156.109, -73.032, -49.226, 39.69, 39.358, -32.688]
  Call Extruder(197.45414)
  MoveL 4234 to (225.5, 35.39, 69.25) mm, rotated rx 180 ry 0 rz 180 deg; joints [-156.117, -73.07, -49.143, 39.714, 39.32, -32.725]
  MoveL 4235 to (225.5, 35.39, 69.25) mm, rotated rx 180 ry 0 rz 180 deg; joints [-156.117, -73.07, -49.143, 39.714, 39.32, -32.725]
  Call Extruder(197.61369)
  MoveL 4236 to (225.8, 35.44, 69.25) mm, rotated rx 180 ry 0 rz 180 deg; joints [-156.125, -73.108, -49.06, 39.739, 39.281, -32.762]
  MoveL 4237 to (225.8, 35.44, 69.25) mm, rotated rx 180 ry 0 rz 180 deg; joints [-156.125, -73.108, -49.06, 39.739, 39.281, -32.762]
  Call Extruder(197.77397)
  MoveL 4238 to (226.11, 35.49, 69.25) mm, rotated rx 180 ry 0 rz 180 deg; joints [-156.133, -73.146, -48.978, 39.763, 39.242, -32.799]
  MoveL 4239 to (226.11, 35.49, 69.25) mm, rotated rx 180 ry 0 rz 180 deg; joints [-156.133, -73.146, -48.978, 39.763, 39.242, -32.799]
  Call Extruder(197.93497)
  MoveL 4240 to (226.41, 35.54, 69.25) mm, rotated rx 180 ry 0 rz -180 deg; joints [-156.141, -73.184, -48.895, 39.788, 39.203, -32.836]
  MoveL 4241 to (226.41, 35.54, 69.25) mm, rotated rx 180 ry 0 rz -180 deg; joints [-156.141, -73.184, -48.895, 39.788, 39.203, -32.836]
  Call Extruder(198.09670)
  MoveL 4242 to (226.72, 35.59, 69.25) mm, rotated rx -180 ry 0 rz 180 deg; joints [-156.149, -73.222, -48.811, 39.812, 39.164, -32.874]
  MoveL 4243 to (226.72, 35.59, 69.25) mm, rotated rx -180 ry 0 rz 180 deg; joints [-156.149, -73.222, -48.811, 39.812, 39.164, -32.874]
  Call Extruder(198.25916)
  MoveL 4244 to (227.03, 35.63, 69.25) mm, rotated rx 180 ry 0 rz -180 deg; joints [-156.157, -73.26, -48.728, 39.837, 39.125, -32.911]
  MoveL 4245 to (227.03, 35.63, 69.25) mm, rotated rx 180 ry 0 rz -180 deg; joints [-156.157, -73.26, -48.728, 39.837, 39.125, -32.911]
  Call Extruder(198.39309)
  MoveL 4246 to (227.28, 35.68, 69.25) mm, rotated rx 180 ry 0 rz 180 deg; joints [-156.162, -73.292, -48.659, 39.859, 39.093, -32.943]
  MoveL 4247 to (227.28, 35.68, 69.25) mm, rotated rx 180 ry 0 rz 180 deg; joints [-156.162, -73.292, -48.659, 39.859, 39.093, -32.943]
  Call Extruder(198.52763)
  MoveL 4248 to (227.52, 35.73, 69.25) mm, rotated rx 180 ry 0 rz -180 deg; joints [-156.168, -73.324, -48.59, 39.882, 39.061, -32.976]
  MoveL 4249 to (227.52, 35.73, 69.25) mm, rotated rx 180 ry 0 rz -180 deg; joints [-156.168, -73.324, -48.59, 39.882, 39.061, -32.976]
  Call Extruder(198.66277)
  MoveL 4250 to (227.77, 35.78, 69.25) mm, rotated rx -180 ry 0 rz 180 deg; joints [-156.173, -73.355, -48.521, 39.904, 39.03, -33.008]
  MoveL 4251 to (227.77, 35.78, 69.25) mm, rotated rx -180 ry 0 rz 180 deg; joints [-156.173, -73.355, -48.521, 39.904, 39.03, -33.008]
  Call Extruder(198.79853)
  MoveL 4252 to (228.02, 35.83, 69.25) mm, rotated rx 180 ry 0 rz 180 deg; joints [-156.179, -73.387, -48.451, 39.926, 38.998, -33.041]
  MoveL 4253 to (228.02, 35.83, 69.25) mm, rotated rx 180 ry 0 rz 180 deg; joints [-156.179, -73.387, -48.451, 39.926, 38.998, -33.041]
  Call Extruder(198.93490)
  MoveL 4254 to (228.27, 35.88, 69.25) mm, rotated rx 180 ry 0 rz 180 deg; joints [-156.185, -73.419, -48.382, 39.949, 38.966, -33.073]
  MoveL 4255 to (228.27, 35.88, 69.25) mm, rotated rx 180 ry 0 rz 180 deg; joints [-156.185, -73.419, -48.382, 39.949, 38.966, -33.073]
  Call Extruder(199.07188)
  MoveL 4256 to (228.52, 35.93, 69.25) mm, rotated rx -180 ry 0 rz 180 deg; joints [-156.19, -73.451, -48.313, 39.971, 38.934, -33.106]
  MoveL 4257 to (228.52, 35.93, 69.25) mm, rotated rx -180 ry 0 rz 180 deg; joints [-156.19, -73.451, -48.313, 39.971, 38.934, -33.106]
  Call Extruder(199.20947)
  MoveL 4258 to (228.77, 35.98, 69.25) mm, rotated rx 180 ry 0 rz 180 deg; joints [-156.196, -73.483, -48.243, 39.994, 38.903, -33.139]
  MoveL 4259 to (228.77, 35.98, 69.25) mm, rotated rx 180 ry 0 rz 180 deg; joints [-156.196, -73.483, -48.243, 39.994, 38.903, -33.139]
  Call Extruder(199.32318)
  MoveL 4260 to (228.97, 36.03, 69.25) mm, rotated rx 180 ry 0 rz 180 deg; joints [-156.2, -73.509, -48.186, 40.013, 38.876, -33.166]
  MoveL 4261 to (228.97, 36.03, 69.25) mm, rotated rx 180 ry 0 rz 180 deg; joints [-156.2, -73.509, -48.186, 40.013, 38.876, -33.166]
  Call Extruder(199.43735)
  MoveL 4262 to (229.18, 36.07, 69.25) mm, rotated rx -180 ry 0 rz 180 deg; joints [-156.204, -73.536, -48.128, 40.032, 38.85, -33.194]
  MoveL 4263 to (229.18, 36.07, 69.25) mm, rotated rx -180 ry 0 rz 180 deg; joints [-156.204, -73.536, -48.128, 40.032, 38.85, -33.194]
  Call Extruder(199.55198)
  MoveL 4264 to (229.38, 36.12, 69.25) mm, rotated rx 180 ry 0 rz 180 deg; joints [-156.208, -73.562, -48.07, 40.052, 38.824, -33.221]
  MoveL 4265 to (229.38, 36.12, 69.25) mm, rotated rx 180 ry 0 rz 180 deg; joints [-156.208, -73.562, -48.07, 40.052, 38.824, -33.221]
  Call Extruder(199.66705)
  MoveL 4266 to (229.59, 36.16, 69.25) mm, rotated rx 180 ry 0 rz -180 deg; joints [-156.212, -73.588, -48.013, 40.071, 38.798, -33.249]
  MoveL 4267 to (229.59, 36.16, 69.25) mm, rotated rx 180 ry 0 rz -180 deg; joints [-156.212, -73.588, -48.013, 40.071, 38.798, -33.249]
  Call Extruder(199.78928)
  MoveL 4268 to (229.8, 36.22, 69.25) mm, rotated rx 180 ry 0 rz 180 deg; joints [-156.216, -73.617, -47.951, 40.093, 38.771, -33.279]
  MoveL 4269 to (229.8, 36.22, 69.25) mm, rotated rx 180 ry 0 rz 180 deg; joints [-156.216, -73.617, -47.951, 40.093, 38.771, -33.279]
  Call Extruder(199.91895)
  MoveL 4270 to (230.02, 36.28, 69.25) mm, rotated rx 180 ry 0 rz -180 deg; joints [-156.219, -73.647, -47.886, 40.117, 38.742, -33.313]
  MoveL 4271 to (230.02, 36.28, 69.25) mm, rotated rx 180 ry 0 rz -180 deg; joints [-156.219, -73.647, -47.886, 40.117, 38.742, -33.313]
  Call Extruder(200.04918)
  MoveL 4272 to (230.25, 36.35, 69.25) mm, rotated rx -180 ry 0 rz 180 deg; joints [-156.221, -73.677, -47.82, 40.142, 38.714, -33.346]
  MoveL 4273 to (230.25, 36.35, 69.25) mm, rotated rx -180 ry 0 rz 180 deg; joints [-156.221, -73.677, -47.82, 40.142, 38.714, -33.346]
  Call Extruder(200.17998)
  MoveL 4274 to (230.47, 36.42, 69.25) mm, rotated rx -180 ry 0 rz 180 deg; joints [-156.224, -73.707, -47.755, 40.167, 38.685, -33.38]
  MoveL 4275 to (230.47, 36.42, 69.25) mm, rotated rx -180 ry 0 rz 180 deg; joints [-156.224, -73.707, -47.755, 40.167, 38.685, -33.38]
  Call Extruder(200.31134)
  MoveL 4276 to (230.69, 36.49, 69.25) mm, rotated rx -180 ry 0 rz 180 deg; joints [-156.227, -73.737, -47.689, 40.192, 38.656, -33.414]
  MoveL 4277 to (230.69, 36.49, 69.25) mm, rotated rx -180 ry 0 rz 180 deg; joints [-156.227, -73.737, -47.689, 40.192, 38.656, -33.414]
  Call Extruder(200.42676)
  MoveL 4278 to (230.89, 36.55, 69.25) mm, rotated rx 180 ry 0 rz 180 deg; joints [-156.229, -73.764, -47.632, 40.214, 38.631, -33.444]
  MoveL 4279 to (230.89, 36.55, 69.25) mm, rotated rx 180 ry 0 rz 180 deg; joints [-156.229, -73.764, -47.632, 40.214, 38.631, -33.444]
  Call Extruder(200.54265)
  MoveL 4280 to (231.08, 36.61, 69.25) mm, rotated rx 180 ry 0 rz -180 deg; joints [-156.231, -73.79, -47.574, 40.236, 38.607, -33.474]
  MoveL 4281 to (231.08, 36.61, 69.25) mm, rotated rx 180 ry 0 rz -180 deg; joints [-156.231, -73.79, -47.574, 40.236, 38.607, -33.474]
  Call Extruder(200.65547)
  MoveL 4282 to (231.27, 36.68, 69.25) mm, rotated rx 180 ry 0 rz 180 deg; joints [-156.233, -73.816, -47.518, 40.258, 38.582, -33.503]
  MoveL 4283 to (231.27, 36.68, 69.25) mm, rotated rx 180 ry 0 rz 180 deg; joints [-156.233, -73.816, -47.518, 40.258, 38.582, -33.503]
  Call Extruder(200.76517)
  MoveL 4284 to (231.45, 36.73, 69.25) mm, rotated rx 180 ry 0 rz -180 deg; joints [-156.235, -73.841, -47.464, 40.279, 38.559, -33.531]
  MoveL 4285 to (231.45, 36.73, 69.25) mm, rotated rx 180 ry 0 rz -180 deg; joints [-156.235, -73.841, -47.464, 40.279, 38.559, -33.531]
  Call Extruder(200.87528)
  MoveL 4286 to (231.64, 36.79, 69.25) mm, rotated rx 180 ry 0 rz 180 deg; joints [-156.237, -73.866, -47.41, 40.3, 38.536, -33.559]
  MoveL 4287 to (231.64, 36.79, 69.25) mm, rotated rx 180 ry 0 rz 180 deg; joints [-156.237, -73.866, -47.41, 40.3, 38.536, -33.559]
  Call Extruder(201.05724)
  MoveL 4288 to (231.93, 36.91, 69.25) mm, rotated rx 180 ry 0 rz 180 deg; joints [-156.238, -73.907, -47.32, 40.339, 38.498, -33.609]
  MoveL 4289 to (231.93, 36.91, 69.25) mm, rotated rx 180 ry 0 rz 180 deg; joints [-156.238, -73.907, -47.32, 40.339, 38.498, -33.609]
  Call Extruder(201.23996)
  MoveL 4290 to (232.22, 37.03, 69.25) mm, rotated rx 180 ry 0 rz 180 deg; joints [-156.238, -73.949, -47.23, 40.377, 38.461, -33.659]
  MoveL 4291 to (232.22, 37.03, 69.25) mm, rotated rx 180 ry 0 rz 180 deg; joints [-156.238, -73.949, -47.23, 40.377, 38.461, -33.659]
  Call Extruder(201.41037)
  MoveL 4292 to (232.49, 37.15, 69.25) mm, rotated rx -180 ry 0 rz 180 deg; joints [-156.239, -73.987, -47.146, 40.414, 38.426, -33.705]
  MoveL 4293 to (232.49, 37.15, 69.25) mm, rotated rx -180 ry 0 rz 180 deg; joints [-156.239, -73.987, -47.146, 40.414, 38.426, -33.705]
  Call Extruder(201.56837)
  MoveL 4294 to (232.74, 37.26, 69.25) mm, rotated rx 180 ry 0 rz -180 deg; joints [-156.239, -74.023, -47.069, 40.447, 38.395, -33.749]
  MoveL 4295 to (232.74, 37.26, 69.25) mm, rotated rx 180 ry 0 rz -180 deg; joints [-156.239, -74.023, -47.069, 40.447, 38.395, -33.749]
  Call Extruder(201.72697)
  MoveL 4296 to (232.99, 37.36, 69.25) mm, rotated rx 180 ry 0 rz -180 deg; joints [-156.239, -74.059, -46.991, 40.481, 38.363, -33.792]
  MoveL 4297 to (232.99, 37.36, 69.25) mm, rotated rx 180 ry 0 rz -180 deg; joints [-156.239, -74.059, -46.991, 40.481, 38.363, -33.792]
  Call Extruder(201.93314)
  MoveL 4298 to (233.29, 37.54, 69.25) mm, rotated rx 180 ry 0 rz 180 deg; joints [-156.236, -74.105, -46.891, 40.53, 38.324, -33.852]
  MoveL 4299 to (233.29, 37.54, 69.25) mm, rotated rx 180 ry 0 rz 180 deg; joints [-156.236, -74.105, -46.891, 40.53, 38.324, -33.852]
  Call Extruder(202.14008)
  MoveL 4300 to (233.6, 37.71, 69.25) mm, rotated rx -180 ry 0 rz 180 deg; joints [-156.232, -74.151, -46.791, 40.58, 38.285, -33.913]
  MoveL 4301 to (233.6, 37.71, 69.25) mm, rotated rx -180 ry 0 rz 180 deg; joints [-156.232, -74.151, -46.791, 40.58, 38.285, -33.913]
  Call Extruder(202.34781)
  MoveL 4302 to (233.9, 37.89, 69.25) mm, rotated rx 180 ry 0 rz 180 deg; joints [-156.228, -74.197, -46.691, 40.629, 38.246, -33.973]
  MoveL 4303 to (233.9, 37.89, 69.25) mm, rotated rx 180 ry 0 rz 180 deg; joints [-156.228, -74.197, -46.691, 40.629, 38.246, -33.973]
  Call Extruder(202.55631)
  MoveL 4304 to (234.21, 38.06, 69.25) mm, rotated rx 180 ry 0 rz 180 deg; joints [-156.224, -74.244, -46.591, 40.679, 38.207, -34.034]
  MoveL 4305 to (234.21, 38.06, 69.25) mm, rotated rx 180 ry 0 rz 180 deg; joints [-156.224, -74.244, -46.591, 40.679, 38.207, -34.034]
  Call Extruder(202.73585)
  MoveL 4306 to (234.45, 38.24, 69.25) mm, rotated rx 180 ry 0 rz -180 deg; joints [-156.218, -74.283, -46.506, 40.725, 38.176, -34.089]
  MoveL 4307 to (234.45, 38.24, 69.25) mm, rotated rx 180 ry 0 rz -180 deg; joints [-156.218, -74.283, -46.506, 40.725, 38.176, -34.089]
  Call Extruder(203.06927)
  MoveL 4308 to (234.9, 38.57, 69.25) mm, rotated rx 180 ry 0 rz 180 deg; joints [-156.206, -74.356, -46.348, 40.811, 38.119, -34.191]
  MoveL 4309 to (234.9, 38.57, 69.25) mm, rotated rx 180 ry 0 rz 180 deg; joints [-156.206, -74.356, -46.348, 40.811, 38.119, -34.191]
  Call Extruder(203.40387)
  MoveL 4310 to (235.35, 38.9, 69.25) mm, rotated rx -180 ry 0 rz -180 deg; joints [-156.195, -74.429, -46.19, 40.898, 38.061, -34.293]
  Call Extruder(204.23182)
  MoveL 4311 to (236.39, 39.81, 69.25) mm, rotated rx 180 ry 0 rz 180 deg; joints [-156.154, -74.606, -45.808, 41.126, 37.929, -34.556]
  Call Extruder(205.05976)
  MoveL 4312 to (237.3, 40.85, 69.25) mm, rotated rx 180 ry 0 rz 180 deg; joints [-156.097, -74.776, -45.441, 41.369, 37.814, -34.827]
  Call Extruder(205.22706)
  MoveL 4313 to (237.47, 41.07, 69.25) mm, rotated rx 180 ry 0 rz 180 deg; joints [-156.083, -74.809, -45.371, 41.42, 37.793, -34.883]
  MoveL 4314 to (237.47, 41.07, 69.25) mm, rotated rx 180 ry 0 rz 180 deg; joints [-156.083, -74.809, -45.371, 41.42, 37.793, -34.883]
  Call Extruder(205.56048)
  MoveL 4315 to (237.8, 41.52, 69.25) mm, rotated rx 180 ry 0 rz -180 deg; joints [-156.055, -74.874, -45.229, 41.521, 37.752, -34.994]
  MoveL 4316 to (237.8, 41.52, 69.25) mm, rotated rx 180 ry 0 rz -180 deg; joints [-156.055, -74.874, -45.229, 41.521, 37.752, -34.994]
  Call Extruder(205.89270)
  MoveL 4317 to (238.12, 41.98, 69.25) mm, rotated rx 180 ry 0 rz -180 deg; joints [-156.028, -74.941, -45.086, 41.624, 37.711, -35.106]
  MoveL 4318 to (238.12, 41.98, 69.25) mm, rotated rx 180 ry 0 rz -180 deg; joints [-156.028, -74.941, -45.086, 41.624, 37.711, -35.106]
  Call Extruder(206.01040)
  MoveL 4319 to (238.22, 42.15, 69.25) mm, rotated rx 180 ry 0 rz 180 deg; joints [-156.016, -74.963, -45.039, 41.66, 37.698, -35.145]
  MoveL 4320 to (238.22, 42.15, 69.25) mm, rotated rx 180 ry 0 rz 180 deg; joints [-156.016, -74.963, -45.039, 41.66, 37.698, -35.145]
  Call Extruder(206.21813)
  MoveL 4321 to (238.4, 42.45, 69.25) mm, rotated rx 180 ry 0 rz -180 deg; joints [-155.996, -75.002, -44.955, 41.726, 37.676, -35.216]
  MoveL 4322 to (238.4, 42.45, 69.25) mm, rotated rx 180 ry 0 rz -180 deg; joints [-155.996, -75.002, -44.955, 41.726, 37.676, -35.216]
  Call Extruder(206.42507)
  MoveL 4323 to (238.57, 42.75, 69.25) mm, rotated rx -180 ry 0 rz 180 deg; joints [-155.976, -75.041, -44.871, 41.792, 37.654, -35.286]
  MoveL 4324 to (238.57, 42.75, 69.25) mm, rotated rx -180 ry 0 rz 180 deg; joints [-155.976, -75.041, -44.871, 41.792, 37.654, -35.286]
  Call Extruder(206.63124)
  MoveL 4325 to (238.75, 43.06, 69.25) mm, rotated rx 180 ry 0 rz 180 deg; joints [-155.956, -75.08, -44.787, 41.858, 37.633, -35.356]
  MoveL 4326 to (238.75, 43.06, 69.25) mm, rotated rx 180 ry 0 rz 180 deg; joints [-155.956, -75.08, -44.787, 41.858, 37.633, -35.356]
  Call Extruder(206.81293)
  MoveL 4327 to (238.89, 43.33, 69.25) mm, rotated rx 180 ry 0 rz 180 deg; joints [-155.937, -75.113, -44.715, 41.917, 37.615, -35.419]
  MoveL 4328 to (238.89, 43.33, 69.25) mm, rotated rx 180 ry 0 rz 180 deg; joints [-155.937, -75.113, -44.715, 41.917, 37.615, -35.419]
  Call Extruder(206.97094)
  MoveL 4329 to (239, 43.58, 69.25) mm, rotated rx -180 ry 0 rz -180 deg; joints [-155.919, -75.141, -44.656, 41.968, 37.602, -35.473]
  MoveL 4330 to (239, 43.58, 69.25) mm, rotated rx -180 ry 0 rz -180 deg; joints [-155.919, -75.141, -44.656, 41.968, 37.602, -35.473]
  Call Extruder(207.12835)
  MoveL 4331 to (239.11, 43.83, 69.25) mm, rotated rx -180 ry 0 rz -180 deg; joints [-155.901, -75.168, -44.597, 42.02, 37.589, -35.526]
  MoveL 4332 to (239.11, 43.83, 69.25) mm, rotated rx -180 ry 0 rz -180 deg; joints [-155.901, -75.168, -44.597, 42.02, 37.589, -35.526]
  Call Extruder(207.31106)
  MoveL 4333 to (239.23, 44.12, 69.25) mm, rotated rx -180 ry 0 rz 180 deg; joints [-155.879, -75.2, -44.529, 42.08, 37.574, -35.589]
  MoveL 4334 to (239.23, 44.12, 69.25) mm, rotated rx -180 ry 0 rz 180 deg; joints [-155.879, -75.2, -44.529, 42.08, 37.574, -35.589]
  Call Extruder(207.49302)
  MoveL 4335 to (239.35, 44.42, 69.25) mm, rotated rx 180 ry 0 rz -180 deg; joints [-155.858, -75.232, -44.46, 42.14, 37.56, -35.651]
  MoveL 4336 to (239.35, 44.42, 69.25) mm, rotated rx 180 ry 0 rz -180 deg; joints [-155.858, -75.232, -44.46, 42.14, 37.56, -35.651]
  Call Extruder(207.64035)
  MoveL 4337 to (239.44, 44.66, 69.25) mm, rotated rx 180 ry 0 rz -180 deg; joints [-155.84, -75.257, -44.406, 42.189, 37.549, -35.702]
  MoveL 4338 to (239.44, 44.66, 69.25) mm, rotated rx 180 ry 0 rz -180 deg; joints [-155.84, -75.257, -44.406, 42.189, 37.549, -35.702]
  Call Extruder(207.75359)
  MoveL 4339 to (239.5, 44.85, 69.25) mm, rotated rx 180 ry 0 rz 180 deg; joints [-155.826, -75.275, -44.366, 42.227, 37.541, -35.741]
  MoveL 4340 to (239.5, 44.85, 69.25) mm, rotated rx 180 ry 0 rz 180 deg; joints [-155.826, -75.275, -44.366, 42.227, 37.541, -35.741]
  Call Extruder(207.86638)
  MoveL 4341 to (239.56, 45.03, 69.25) mm, rotated rx 180 ry 0 rz 180 deg; joints [-155.811, -75.294, -44.327, 42.265, 37.534, -35.779]
  MoveL 4342 to (239.56, 45.03, 69.25) mm, rotated rx 180 ry 0 rz 180 deg; joints [-155.811, -75.294, -44.327, 42.265, 37.534, -35.779]
  Call Extruder(207.97872)
  MoveL 4343 to (239.62, 45.22, 69.25) mm, rotated rx 180 ry 0 rz -180 deg; joints [-155.797, -75.312, -44.287, 42.302, 37.527, -35.818]
  MoveL 4344 to (239.62, 45.22, 69.25) mm, rotated rx 180 ry 0 rz -180 deg; joints [-155.797, -75.312, -44.287, 42.302, 37.527, -35.818]
  Call Extruder(208.09063)
  MoveL 4345 to (239.68, 45.41, 69.25) mm, rotated rx -180 ry 0 rz 180 deg; joints [-155.783, -75.331, -44.247, 42.34, 37.519, -35.856]
  MoveL 4346 to (239.68, 45.41, 69.25) mm, rotated rx -180 ry 0 rz 180 deg; joints [-155.783, -75.331, -44.247, 42.34, 37.519, -35.856]
  Call Extruder(208.21203)
  MoveL 4347 to (239.75, 45.62, 69.25) mm, rotated rx 180 ry 0 rz 180 deg; joints [-155.767, -75.351, -44.204, 42.381, 37.512, -35.899]
  MoveL 4348 to (239.75, 45.62, 69.25) mm, rotated rx 180 ry 0 rz 180 deg; joints [-155.767, -75.351, -44.204, 42.381, 37.512, -35.899]
  Call Extruder(208.34282)
  MoveL 4349 to (239.81, 45.84, 69.25) mm, rotated rx 180 ry 0 rz 180 deg; joints [-155.75, -75.372, -44.158, 42.426, 37.504, -35.944]
  MoveL 4350 to (239.81, 45.84, 69.25) mm, rotated rx 180 ry 0 rz 180 deg; joints [-155.75, -75.372, -44.158, 42.426, 37.504, -35.944]
  Call Extruder(208.47304)
  MoveL 4351 to (239.88, 46.06, 69.25) mm, rotated rx -180 ry 0 rz 180 deg; joints [-155.733, -75.394, -44.113, 42.47, 37.496, -35.989]
  MoveL 4352 to (239.88, 46.06, 69.25) mm, rotated rx -180 ry 0 rz 180 deg; joints [-155.733, -75.394, -44.113, 42.47, 37.496, -35.989]
  Call Extruder(208.60270)
  MoveL 4353 to (239.95, 46.29, 69.25) mm, rotated rx 180 ry 0 rz 180 deg; joints [-155.715, -75.415, -44.066, 42.515, 37.488, -36.035]
  MoveL 4354 to (239.95, 46.29, 69.25) mm, rotated rx 180 ry 0 rz 180 deg; joints [-155.715, -75.415, -44.066, 42.515, 37.488, -36.035]
  Call Extruder(208.73180)
  MoveL 4355 to (240.02, 46.51, 69.25) mm, rotated rx 180 ry 0 rz 180 deg; joints [-155.698, -75.436, -44.02, 42.559, 37.48, -36.08]
  MoveL 4356 to (240.02, 46.51, 69.25) mm, rotated rx 180 ry 0 rz 180 deg; joints [-155.698, -75.436, -44.02, 42.559, 37.48, -36.08]
  Call Extruder(208.84685)
  MoveL 4357 to (240.06, 46.72, 69.25) mm, rotated rx 180 ry 0 rz -180 deg; joints [-155.682, -75.454, -43.983, 42.599, 37.474, -36.12]
  MoveL 4358 to (240.06, 46.72, 69.25) mm, rotated rx 180 ry 0 rz -180 deg; joints [-155.682, -75.454, -43.983, 42.599, 37.474, -36.12]
  Call Extruder(208.96145)
  MoveL 4359 to (240.11, 46.92, 69.25) mm, rotated rx 180 ry 0 rz 180 deg; joints [-155.665, -75.471, -43.945, 42.638, 37.469, -36.159]
  MoveL 4360 to (240.11, 46.92, 69.25) mm, rotated rx 180 ry 0 rz 180 deg; joints [-155.665, -75.471, -43.945, 42.638, 37.469, -36.159]
  Call Extruder(209.07560)
  MoveL 4361 to (240.15, 47.12, 69.25) mm, rotated rx 180 ry 0 rz 180 deg; joints [-155.649, -75.489, -43.908, 42.677, 37.464, -36.199]
  MoveL 4362 to (240.15, 47.12, 69.25) mm, rotated rx 180 ry 0 rz 180 deg; joints [-155.649, -75.489, -43.908, 42.677, 37.464, -36.199]
  Call Extruder(209.18930)
  MoveL 4363 to (240.2, 47.33, 69.25) mm, rotated rx 180 ry 0 rz 180 deg; joints [-155.633, -75.506, -43.87, 42.717, 37.459, -36.238]
  MoveL 4364 to (240.2, 47.33, 69.25) mm, rotated rx 180 ry 0 rz 180 deg; joints [-155.633, -75.506, -43.87, 42.717, 37.459, -36.238]
  Call Extruder(209.31471)
  MoveL 4365 to (240.24, 47.55, 69.25) mm, rotated rx 180 ry 0 rz 180 deg; joints [-155.614, -75.526, -43.829, 42.76, 37.454, -36.282]
  MoveL 4366 to (240.24, 47.55, 69.25) mm, rotated rx 180 ry 0 rz 180 deg; joints [-155.614, -75.526, -43.829, 42.76, 37.454, -36.282]
  Call Extruder(209.45169)
  MoveL 4367 to (240.29, 47.8, 69.25) mm, rotated rx 180 ry 0 rz 180 deg; joints [-155.594, -75.546, -43.785, 42.808, 37.448, -36.33]
  MoveL 4368 to (240.29, 47.8, 69.25) mm, rotated rx 180 ry 0 rz 180 deg; joints [-155.594, -75.546, -43.785, 42.808, 37.448, -36.33]
  Call Extruder(209.58805)
  MoveL 4369 to (240.34, 48.05, 69.25) mm, rotated rx 180 ry 0 rz 180 deg; joints [-155.574, -75.567, -43.74, 42.856, 37.443, -36.377]
  MoveL 4370 to (240.34, 48.05, 69.25) mm, rotated rx 180 ry 0 rz 180 deg; joints [-155.574, -75.567, -43.74, 42.856, 37.443, -36.377]
  Call Extruder(209.72381)
  MoveL 4371 to (240.39, 48.3, 69.25) mm, rotated rx 180 ry 0 rz 180 deg; joints [-155.554, -75.588, -43.695, 42.904, 37.437, -36.425]
  MoveL 4372 to (240.39, 48.3, 69.25) mm, rotated rx 180 ry 0 rz 180 deg; joints [-155.554, -75.588, -43.695, 42.904, 37.437, -36.425]
  Call Extruder(209.85896)
  MoveL 4373 to (240.44, 48.55, 69.25) mm, rotated rx 180 ry 0 rz 180 deg; joints [-155.534, -75.609, -43.651, 42.952, 37.432, -36.473]
  MoveL 4374 to (240.44, 48.55, 69.25) mm, rotated rx 180 ry 0 rz 180 deg; joints [-155.534, -75.609, -43.651, 42.952, 37.432, -36.473]
  Call Extruder(209.99349)
  MoveL 4375 to (240.49, 48.8, 69.25) mm, rotated rx 180 ry 0 rz 180 deg; joints [-155.514, -75.63, -43.606, 43, 37.426, -36.521]
  MoveL 4376 to (240.49, 48.8, 69.25) mm, rotated rx 180 ry 0 rz 180 deg; joints [-155.514, -75.63, -43.606, 43, 37.426, -36.521]
  Call Extruder(210.12742)
  MoveL 4377 to (240.54, 49.05, 69.25) mm, rotated rx -180 ry 0 rz 180 deg; joints [-155.494, -75.651, -43.561, 43.047, 37.421, -36.569]
  MoveL 4378 to (240.54, 49.05, 69.25) mm, rotated rx -180 ry 0 rz 180 deg; joints [-155.494, -75.651, -43.561, 43.047, 37.421, -36.569]
  Call Extruder(210.27529)
  MoveL 4379 to (240.59, 49.33, 69.25) mm, rotated rx -180 ry 0 rz 180 deg; joints [-155.471, -75.673, -43.513, 43.1, 37.415, -36.622]
  MoveL 4380 to (240.59, 49.33, 69.25) mm, rotated rx -180 ry 0 rz 180 deg; joints [-155.471, -75.673, -43.513, 43.1, 37.415, -36.622]
  Call Extruder(210.43703)
  MoveL 4381 to (240.64, 49.63, 69.25) mm, rotated rx -180 ry 0 rz -180 deg; joints [-155.446, -75.697, -43.461, 43.158, 37.41, -36.679]
  MoveL 4382 to (240.64, 49.63, 69.25) mm, rotated rx -180 ry 0 rz -180 deg; joints [-155.446, -75.697, -43.461, 43.158, 37.41, -36.679]
  Call Extruder(210.59805)
  MoveL 4383 to (240.69, 49.94, 69.25) mm, rotated rx -180 ry 0 rz 180 deg; joints [-155.421, -75.722, -43.409, 43.216, 37.405, -36.737]
  MoveL 4384 to (240.69, 49.94, 69.25) mm, rotated rx -180 ry 0 rz 180 deg; joints [-155.421, -75.722, -43.409, 43.216, 37.405, -36.737]
  Call Extruder(210.75834)
  MoveL 4385 to (240.74, 50.24, 69.25) mm, rotated rx 180 ry 0 rz 180 deg; joints [-155.396, -75.746, -43.357, 43.274, 37.4, -36.794]
  MoveL 4386 to (240.74, 50.24, 69.25) mm, rotated rx 180 ry 0 rz 180 deg; joints [-155.396, -75.746, -43.357, 43.274, 37.4, -36.794]
  Call Extruder(210.91790)
  MoveL 4387 to (240.78, 50.55, 69.25) mm, rotated rx 180 ry 0 rz 180 deg; joints [-155.371, -75.77, -43.305, 43.332, 37.395, -36.852]
  MoveL 4388 to (240.78, 50.55, 69.25) mm, rotated rx 180 ry 0 rz 180 deg; joints [-155.371, -75.77, -43.305, 43.332, 37.395, -36.852]
  Call Extruder(211.07673)
  MoveL 4389 to (240.83, 50.86, 69.25) mm, rotated rx 180 ry 0 rz 180 deg; joints [-155.346, -75.795, -43.253, 43.39, 37.39, -36.909]
  MoveL 4390 to (240.83, 50.86, 69.25) mm, rotated rx 180 ry 0 rz 180 deg; joints [-155.346, -75.795, -43.253, 43.39, 37.39, -36.909]
  Call Extruder(211.25540)
  MoveL 4391 to (240.88, 51.2, 69.25) mm, rotated rx 180 ry 0 rz 180 deg; joints [-155.317, -75.821, -43.196, 43.455, 37.385, -36.974]
  MoveL 4392 to (240.88, 51.2, 69.25) mm, rotated rx 180 ry 0 rz 180 deg; joints [-155.317, -75.821, -43.196, 43.455, 37.385, -36.974]
  Call Extruder(211.45384)
  MoveL 4393 to (240.92, 51.59, 69.25) mm, rotated rx 180 ry 0 rz -180 deg; joints [-155.285, -75.85, -43.134, 43.527, 37.38, -37.045]
  MoveL 4394 to (240.92, 51.59, 69.25) mm, rotated rx 180 ry 0 rz -180 deg; joints [-155.285, -75.85, -43.134, 43.527, 37.38, -37.045]
  Call Extruder(211.65142)
  MoveL 4395 to (240.97, 51.98, 69.25) mm, rotated rx 180 ry 0 rz 180 deg; joints [-155.252, -75.879, -43.072, 43.599, 37.376, -37.116]
  MoveL 4396 to (240.97, 51.98, 69.25) mm, rotated rx 180 ry 0 rz 180 deg; joints [-155.252, -75.879, -43.072, 43.599, 37.376, -37.116]
  Call Extruder(211.84813)
  MoveL 4397 to (241.02, 52.36, 69.25) mm, rotated rx 180 ry 0 rz -180 deg; joints [-155.22, -75.908, -43.01, 43.672, 37.371, -37.188]
  MoveL 4398 to (241.02, 52.36, 69.25) mm, rotated rx 180 ry 0 rz -180 deg; joints [-155.22, -75.908, -43.01, 43.672, 37.371, -37.188]
  Call Extruder(212.04396)
  MoveL 4399 to (241.06, 52.75, 69.25) mm, rotated rx 180 ry 0 rz 180 deg; joints [-155.188, -75.937, -42.948, 43.744, 37.367, -37.259]
  MoveL 4400 to (241.06, 52.75, 69.25) mm, rotated rx 180 ry 0 rz 180 deg; joints [-155.188, -75.937, -42.948, 43.744, 37.367, -37.259]
  Call Extruder(212.33940)
  MoveL 4401 to (241.11, 53.34, 69.25) mm, rotated rx -180 ry 0 rz 180 deg; joints [-155.138, -75.979, -42.859, 43.852, 37.363, -37.365]
  MoveL 4402 to (241.11, 53.34, 69.25) mm, rotated rx -180 ry 0 rz 180 deg; joints [-155.138, -75.979, -42.859, 43.852, 37.363, -37.365]
  Call Extruder(212.63351)
  MoveL 4403 to (241.16, 53.93, 69.25) mm, rotated rx -180 ry 0 rz 180 deg; joints [-155.088, -76.02, -42.77, 43.961, 37.36, -37.471]
  MoveL 4404 to (241.16, 53.93, 69.25) mm, rotated rx -180 ry 0 rz 180 deg; joints [-155.088, -76.02, -42.77, 43.961, 37.36, -37.471]
  Call Extruder(212.92629)
  MoveL 4405 to (241.2, 54.52, 69.25) mm, rotated rx -180 ry 0 rz 180 deg; joints [-155.038, -76.062, -42.681, 44.069, 37.356, -37.577]
  MoveL 4406 to (241.2, 54.52, 69.25) mm, rotated rx -180 ry 0 rz 180 deg; joints [-155.038, -76.062, -42.681, 44.069, 37.356, -37.577]
  Call Extruder(213.49974)
  MoveL 4407 to (241.25, 55.68, 69.25) mm, rotated rx 180 ry 0 rz 180 deg; joints [-154.938, -76.139, -42.517, 44.279, 37.355, -37.781]
  MoveL 4408 to (241.25, 55.68, 69.25) mm, rotated rx 180 ry 0 rz 180 deg; joints [-154.938, -76.139, -42.517, 44.279, 37.355, -37.781]
  Call Extruder(214.21357)
  MoveL 4409 to (241.29, 57.14, 69.25) mm, rotated rx 180 ry 0 rz 180 deg; joints [-154.812, -76.233, -42.316, 44.541, 37.356, -38.034]
  Call Extruder(256.27845)
  MoveL 4410 to (241.29, 142.86, 69.25) mm, rotated rx -180 ry 0 rz 180 deg; joints [-147.778, -83.221, -27.726, 60.438, 37.807, -54.325]
  Call Extruder(256.70688)
  MoveL 4411 to (241.27, 143.73, 69.25) mm, rotated rx 180 ry 0 rz 180 deg; joints [-147.711, -83.312, -27.538, 60.609, 37.814, -54.512]
  MoveL 4412 to (241.27, 143.73, 69.25) mm, rotated rx 180 ry 0 rz 180 deg; joints [-147.711, -83.312, -27.538, 60.609, 37.814, -54.512]
  Call Extruder(257.28033)
  MoveL 4413 to (241.22, 144.9, 69.25) mm, rotated rx -180 ry 0 rz -180 deg; joints [-147.62, -83.432, -27.294, 60.836, 37.827, -54.757]
  MoveL 4414 to (241.22, 144.9, 69.25) mm, rotated rx -180 ry 0 rz -180 deg; joints [-147.62, -83.432, -27.294, 60.836, 37.827, -54.757]
  Call Extruder(257.71467)
  MoveL 4415 to (241.18, 145.77, 69.25) mm, rotated rx 180 ry 0 rz 180 deg; joints [-147.551, -83.52, -27.113, 61.004, 37.839, -54.94]
  MoveL 4416 to (241.18, 145.77, 69.25) mm, rotated rx 180 ry 0 rz 180 deg; joints [-147.551, -83.52, -27.113, 61.004, 37.839, -54.94]
  Call Extruder(258.00878)
  MoveL 4417 to (241.13, 146.36, 69.25) mm, rotated rx -180 ry 0 rz -180 deg; joints [-147.504, -83.577, -26.996, 61.115, 37.849, -55.06]
  MoveL 4418 to (241.13, 146.36, 69.25) mm, rotated rx -180 ry 0 rz -180 deg; joints [-147.504, -83.577, -26.996, 61.115, 37.849, -55.06]
  Call Extruder(258.30422)
  MoveL 4419 to (241.09, 146.95, 69.25) mm, rotated rx -180 ry 0 rz 180 deg; joints [-147.457, -83.635, -26.878, 61.227, 37.858, -55.18]
  MoveL 4420 to (241.09, 146.95, 69.25) mm, rotated rx -180 ry 0 rz 180 deg; joints [-147.457, -83.635, -26.878, 61.227, 37.858, -55.18]
  Call Extruder(258.55047)
  MoveL 4421 to (241.04, 147.44, 69.25) mm, rotated rx -180 ry 0 rz 180 deg; joints [-147.417, -83.681, -26.783, 61.318, 37.867, -55.278]
  MoveL 4422 to (241.04, 147.44, 69.25) mm, rotated rx -180 ry 0 rz 180 deg; joints [-147.417, -83.681, -26.783, 61.318, 37.867, -55.278]
  Call Extruder(258.74718)
  MoveL 4423 to (240.99, 147.83, 69.25) mm, rotated rx 180 ry 0 rz 180 deg; joints [-147.386, -83.717, -26.711, 61.389, 37.876, -55.354]
  MoveL 4424 to (240.99, 147.83, 69.25) mm, rotated rx 180 ry 0 rz 180 deg; joints [-147.386, -83.717, -26.711, 61.389, 37.876, -55.354]
  Call Extruder(258.94475)
  MoveL 4425 to (240.95, 148.22, 69.25) mm, rotated rx 180 ry 0 rz 180 deg; joints [-147.354, -83.752, -26.639, 61.46, 37.884, -55.43]
  MoveL 4426 to (240.95, 148.22, 69.25) mm, rotated rx 180 ry 0 rz 180 deg; joints [-147.354, -83.752, -26.639, 61.46, 37.884, -55.43]
  Call Extruder(259.14319)
  MoveL 4427 to (240.9, 148.6, 69.25) mm, rotated rx 180 ry 0 rz -180 deg; joints [-147.322, -83.788, -26.566, 61.531, 37.892, -55.506]
  MoveL 4428 to (240.9, 148.6, 69.25) mm, rotated rx 180 ry 0 rz -180 deg; joints [-147.322, -83.788, -26.566, 61.531, 37.892, -55.506]
  Call Extruder(259.34250)
  MoveL 4429 to (240.86, 148.99, 69.25) mm, rotated rx 180 ry 0 rz 180 deg; joints [-147.291, -83.824, -26.493, 61.602, 37.901, -55.583]
  MoveL 4430 to (240.86, 148.99, 69.25) mm, rotated rx 180 ry 0 rz 180 deg; joints [-147.291, -83.824, -26.493, 61.602, 37.901, -55.583]
  Call Extruder(259.50134)
  MoveL 4431 to (240.81, 149.3, 69.25) mm, rotated rx 180 ry 0 rz 180 deg; joints [-147.265, -83.85, -26.44, 61.657, 37.909, -55.64]
  MoveL 4432 to (240.81, 149.3, 69.25) mm, rotated rx 180 ry 0 rz 180 deg; joints [-147.265, -83.85, -26.44, 61.657, 37.909, -55.64]
  Call Extruder(259.66090)
  MoveL 4433 to (240.76, 149.6, 69.25) mm, rotated rx 180 ry 0 rz 180 deg; joints [-147.24, -83.876, -26.387, 61.711, 37.917, -55.697]
  MoveL 4434 to (240.76, 149.6, 69.25) mm, rotated rx 180 ry 0 rz 180 deg; joints [-147.24, -83.876, -26.387, 61.711, 37.917, -55.697]
  Call Extruder(259.82119)
  MoveL 4435 to (240.71, 149.91, 69.25) mm, rotated rx 180 ry 0 rz 180 deg; joints [-147.214, -83.902, -26.333, 61.765, 37.925, -55.755]
  MoveL 4436 to (240.71, 149.91, 69.25) mm, rotated rx 180 ry 0 rz 180 deg; joints [-147.214, -83.902, -26.333, 61.765, 37.925, -55.755]
  Call Extruder(259.98220)
  MoveL 4437 to (240.66, 150.21, 69.25) mm, rotated rx 180 ry 0 rz 180 deg; joints [-147.189, -83.928, -26.28, 61.819, 37.933, -55.812]
  MoveL 4438 to (240.66, 150.21, 69.25) mm, rotated rx 180 ry 0 rz 180 deg; joints [-147.189, -83.928, -26.28, 61.819, 37.933, -55.812]
  Call Extruder(260.14395)
  MoveL 4439 to (240.61, 150.52, 69.25) mm, rotated rx 180 ry 0 rz 180 deg; joints [-147.163, -83.955, -26.226, 61.873, 37.941, -55.87]
  MoveL 4440 to (240.61, 150.52, 69.25) mm, rotated rx 180 ry 0 rz 180 deg; joints [-147.163, -83.955, -26.226, 61.873, 37.941, -55.87]
  Call Extruder(260.30642)
  MoveL 4441 to (240.56, 150.83, 69.25) mm, rotated rx 180 ry 0 rz -180 deg; joints [-147.138, -83.981, -26.172, 61.928, 37.95, -55.928]
  MoveL 4442 to (240.56, 150.83, 69.25) mm, rotated rx 180 ry 0 rz -180 deg; joints [-147.138, -83.981, -26.172, 61.928, 37.95, -55.928]
  Call Extruder(260.44035)
  MoveL 4443 to (240.52, 151.07, 69.25) mm, rotated rx 180 ry 0 rz 180 deg; joints [-147.117, -84.001, -26.131, 61.97, 37.958, -55.973]
  MoveL 4444 to (240.52, 151.07, 69.25) mm, rotated rx 180 ry 0 rz 180 deg; joints [-147.117, -84.001, -26.131, 61.97, 37.958, -55.973]
  Call Extruder(260.57488)
  MoveL 4445 to (240.47, 151.32, 69.25) mm, rotated rx 180 ry 0 rz 180 deg; joints [-147.095, -84.021, -26.091, 62.013, 37.966, -56.017]
  MoveL 4446 to (240.47, 151.32, 69.25) mm, rotated rx 180 ry 0 rz 180 deg; joints [-147.095, -84.021, -26.091, 62.013, 37.966, -56.017]
  Call Extruder(260.71003)
  MoveL 4447 to (240.42, 151.57, 69.25) mm, rotated rx 180 ry 0 rz 180 deg; joints [-147.074, -84.041, -26.051, 62.055, 37.973, -56.062]
  MoveL 4448 to (240.42, 151.57, 69.25) mm, rotated rx 180 ry 0 rz 180 deg; joints [-147.074, -84.041, -26.051, 62.055, 37.973, -56.062]
  Call Extruder(260.84579)
  MoveL 4449 to (240.37, 151.82, 69.25) mm, rotated rx -180 ry 0 rz -180 deg; joints [-147.053, -84.061, -26.01, 62.098, 37.981, -56.107]
  MoveL 4450 to (240.37, 151.82, 69.25) mm, rotated rx -180 ry 0 rz -180 deg; joints [-147.053, -84.061, -26.01, 62.098, 37.981, -56.107]
  Call Extruder(260.98215)
  MoveL 4451 to (240.32, 152.07, 69.25) mm, rotated rx 180 ry 0 rz 180 deg; joints [-147.032, -84.08, -25.969, 62.141, 37.989, -56.152]
  MoveL 4452 to (240.32, 152.07, 69.25) mm, rotated rx 180 ry 0 rz 180 deg; joints [-147.032, -84.08, -25.969, 62.141, 37.989, -56.152]
  Call Extruder(261.11913)
  MoveL 4453 to (240.27, 152.32, 69.25) mm, rotated rx 180 ry 0 rz 180 deg; joints [-147.011, -84.1, -25.929, 62.183, 37.997, -56.197]
  MoveL 4454 to (240.27, 152.32, 69.25) mm, rotated rx 180 ry 0 rz 180 deg; joints [-147.011, -84.1, -25.929, 62.183, 37.997, -56.197]
  Call Extruder(261.25672)
  MoveL 4455 to (240.22, 152.57, 69.25) mm, rotated rx 180 ry 0 rz 180 deg; joints [-146.989, -84.12, -25.888, 62.226, 38.005, -56.242]
  MoveL 4456 to (240.22, 152.57, 69.25) mm, rotated rx 180 ry 0 rz 180 deg; joints [-146.989, -84.12, -25.888, 62.226, 38.005, -56.242]
  Call Extruder(261.37042)
  MoveL 4457 to (240.17, 152.77, 69.25) mm, rotated rx 180 ry 0 rz 180 deg; joints [-146.972, -84.136, -25.855, 62.261, 38.012, -56.278]
  MoveL 4458 to (240.17, 152.77, 69.25) mm, rotated rx 180 ry 0 rz 180 deg; joints [-146.972, -84.136, -25.855, 62.261, 38.012, -56.278]
  Call Extruder(261.48457)
  MoveL 4459 to (240.13, 152.98, 69.25) mm, rotated rx 180 ry 0 rz -180 deg; joints [-146.954, -84.152, -25.823, 62.295, 38.019, -56.314]
  MoveL 4460 to (240.13, 152.98, 69.25) mm, rotated rx 180 ry 0 rz -180 deg; joints [-146.954, -84.152, -25.823, 62.295, 38.019, -56.314]
  Call Extruder(261.59917)
  MoveL 4461 to (240.08, 153.18, 69.25) mm, rotated rx -180 ry 0 rz 180 deg; joints [-146.937, -84.168, -25.791, 62.329, 38.026, -56.35]
  MoveL 4462 to (240.08, 153.18, 69.25) mm, rotated rx -180 ry 0 rz 180 deg; joints [-146.937, -84.168, -25.791, 62.329, 38.026, -56.35]
  Call Extruder(261.71422)
  MoveL 4463 to (240.04, 153.39, 69.25) mm, rotated rx -180 ry 0 rz -180 deg; joints [-146.919, -84.184, -25.759, 62.364, 38.033, -56.386]
  MoveL 4464 to (240.04, 153.39, 69.25) mm, rotated rx -180 ry 0 rz -180 deg; joints [-146.919, -84.184, -25.759, 62.364, 38.033, -56.386]
  Call Extruder(261.83645)
  MoveL 4465 to (239.98, 153.6, 69.25) mm, rotated rx 180 ry 0 rz -180 deg; joints [-146.9, -84.199, -25.729, 62.398, 38.042, -56.422]
  MoveL 4466 to (239.98, 153.6, 69.25) mm, rotated rx 180 ry 0 rz -180 deg; joints [-146.9, -84.199, -25.729, 62.398, 38.042, -56.422]
  Call Extruder(261.96611)
  MoveL 4467 to (239.92, 153.82, 69.25) mm, rotated rx -180 ry 0 rz -180 deg; joints [-146.88, -84.213, -25.7, 62.433, 38.052, -56.457]
  MoveL 4468 to (239.92, 153.82, 69.25) mm, rotated rx -180 ry 0 rz -180 deg; joints [-146.88, -84.213, -25.7, 62.433, 38.052, -56.457]
  Call Extruder(262.09633)
  MoveL 4469 to (239.85, 154.05, 69.25) mm, rotated rx 180 ry 0 rz 180 deg; joints [-146.86, -84.226, -25.672, 62.467, 38.062, -56.492]
  MoveL 4470 to (239.85, 154.05, 69.25) mm, rotated rx 180 ry 0 rz 180 deg; joints [-146.86, -84.226, -25.672, 62.467, 38.062, -56.492]
  Call Extruder(262.22712)
  MoveL 4471 to (239.78, 154.27, 69.25) mm, rotated rx -180 ry 0 rz -180 deg; joints [-146.84, -84.241, -25.643, 62.502, 38.072, -56.527]
  MoveL 4472 to (239.78, 154.27, 69.25) mm, rotated rx -180 ry 0 rz -180 deg; joints [-146.84, -84.241, -25.643, 62.502, 38.072, -56.527]
  Call Extruder(262.35848)
  MoveL 4473 to (239.71, 154.5, 69.25) mm, rotated rx 180 ry 0 rz 180 deg; joints [-146.82, -84.255, -25.614, 62.536, 38.082, -56.562]
  MoveL 4474 to (239.71, 154.5, 69.25) mm, rotated rx 180 ry 0 rz 180 deg; joints [-146.82, -84.255, -25.614, 62.536, 38.082, -56.562]
  Call Extruder(262.47038)
  MoveL 4475 to (239.65, 154.68, 69.25) mm, rotated rx 180 ry 0 rz -180 deg; joints [-146.803, -84.266, -25.591, 62.565, 38.091, -56.591]
  MoveL 4476 to (239.65, 154.68, 69.25) mm, rotated rx 180 ry 0 rz -180 deg; joints [-146.803, -84.266, -25.591, 62.565, 38.091, -56.591]
  Call Extruder(262.58272)
  MoveL 4477 to (239.59, 154.87, 69.25) mm, rotated rx 180 ry 0 rz 180 deg; joints [-146.785, -84.277, -25.568, 62.593, 38.1, -56.62]
  MoveL 4478 to (239.59, 154.87, 69.25) mm, rotated rx 180 ry 0 rz 180 deg; joints [-146.785, -84.277, -25.568, 62.593, 38.1, -56.62]
  Call Extruder(262.69551)
  MoveL 4479 to (239.53, 155.06, 69.25) mm, rotated rx -180 ry 0 rz -180 deg; joints [-146.768, -84.288, -25.546, 62.621, 38.109, -56.648]
  MoveL 4480 to (239.53, 155.06, 69.25) mm, rotated rx -180 ry 0 rz -180 deg; joints [-146.768, -84.288, -25.546, 62.621, 38.109, -56.648]
  Call Extruder(262.80875)
  MoveL 4481 to (239.47, 155.25, 69.25) mm, rotated rx -180 ry 0 rz 180 deg; joints [-146.751, -84.299, -25.523, 62.65, 38.118, -56.677]
  MoveL 4482 to (239.47, 155.25, 69.25) mm, rotated rx -180 ry 0 rz 180 deg; joints [-146.751, -84.299, -25.523, 62.65, 38.118, -56.677]
  Call Extruder(262.92243)
  MoveL 4483 to (239.41, 155.44, 69.25) mm, rotated rx 180 ry 0 rz 180 deg; joints [-146.734, -84.311, -25.5, 62.678, 38.127, -56.706]
  MoveL 4484 to (239.41, 155.44, 69.25) mm, rotated rx 180 ry 0 rz 180 deg; joints [-146.734, -84.311, -25.5, 62.678, 38.127, -56.706]
  Call Extruder(263.10439)
  MoveL 4485 to (239.29, 155.73, 69.25) mm, rotated rx 180 ry 0 rz 180 deg; joints [-146.706, -84.323, -25.474, 62.718, 38.144, -56.744]
  MoveL 4486 to (239.29, 155.73, 69.25) mm, rotated rx 180 ry 0 rz 180 deg; joints [-146.706, -84.323, -25.474, 62.718, 38.144, -56.744]
  Call Extruder(263.28710)
  MoveL 4487 to (239.16, 156.02, 69.25) mm, rotated rx 180 ry 0 rz 180 deg; joints [-146.678, -84.336, -25.448, 62.758, 38.161, -56.783]
  MoveL 4488 to (239.16, 156.02, 69.25) mm, rotated rx 180 ry 0 rz 180 deg; joints [-146.678, -84.336, -25.448, 62.758, 38.161, -56.783]
  Call Extruder(263.45752)
  MoveL 4489 to (239.05, 156.29, 69.25) mm, rotated rx 180 ry 0 rz 180 deg; joints [-146.652, -84.348, -25.425, 62.794, 38.177, -56.818]
  MoveL 4490 to (239.05, 156.29, 69.25) mm, rotated rx 180 ry 0 rz 180 deg; joints [-146.652, -84.348, -25.425, 62.794, 38.177, -56.818]
  Call Extruder(263.61554)
  MoveL 4491 to (238.94, 156.54, 69.25) mm, rotated rx 180 ry 0 rz 180 deg; joints [-146.628, -84.358, -25.404, 62.827, 38.193, -56.85]
  MoveL 4492 to (238.94, 156.54, 69.25) mm, rotated rx 180 ry 0 rz 180 deg; joints [-146.628, -84.358, -25.404, 62.827, 38.193, -56.85]
  Call Extruder(263.77415)
  MoveL 4493 to (238.84, 156.79, 69.25) mm, rotated rx 180 ry 0 rz 180 deg; joints [-146.604, -84.368, -25.383, 62.861, 38.208, -56.882]
  MoveL 4494 to (238.84, 156.79, 69.25) mm, rotated rx 180 ry 0 rz 180 deg; joints [-146.604, -84.368, -25.383, 62.861, 38.208, -56.882]
  Call Extruder(263.98032)
  MoveL 4495 to (238.66, 157.09, 69.25) mm, rotated rx 180 ry 0 rz 180 deg; joints [-146.573, -84.373, -25.374, 62.894, 38.232, -56.91]
  MoveL 4496 to (238.66, 157.09, 69.25) mm, rotated rx 180 ry 0 rz 180 deg; joints [-146.573, -84.373, -25.374, 62.894, 38.232, -56.91]
  Call Extruder(264.18727)
  MoveL 4497 to (238.49, 157.4, 69.25) mm, rotated rx 180 ry 0 rz 180 deg; joints [-146.542, -84.377, -25.364, 62.927, 38.256, -56.939]
  MoveL 4498 to (238.49, 157.4, 69.25) mm, rotated rx 180 ry 0 rz 180 deg; joints [-146.542, -84.377, -25.364, 62.927, 38.256, -56.939]
  Call Extruder(264.39499)
  MoveL 4499 to (238.31, 157.7, 69.25) mm, rotated rx 180 ry 0 rz -180 deg; joints [-146.51, -84.382, -25.355, 62.96, 38.28, -56.968]
  MoveL 4500 to (238.31, 157.7, 69.25) mm, rotated rx 180 ry 0 rz -180 deg; joints [-146.51, -84.382, -25.355, 62.96, 38.28, -56.968]
  Call Extruder(264.60350)
  MoveL 4501 to (238.13, 158.01, 69.25) mm, rotated rx 180 ry 0 rz 180 deg; joints [-146.479, -84.387, -25.346, 62.993, 38.304, -56.996]
  MoveL 4502 to (238.13, 158.01, 69.25) mm, rotated rx 180 ry 0 rz 180 deg; joints [-146.479, -84.387, -25.346, 62.993, 38.304, -56.996]
  Call Extruder(264.78304)
  MoveL 4503 to (237.96, 158.25, 69.25) mm, rotated rx -180 ry 0 rz -180 deg; joints [-146.452, -84.384, -25.351, 63.014, 38.328, -57.011]
  MoveL 4504 to (237.96, 158.25, 69.25) mm, rotated rx -180 ry 0 rz -180 deg; joints [-146.452, -84.384, -25.351, 63.014, 38.328, -57.011]
  Call Extruder(265.11645)
  MoveL 4505 to (237.63, 158.7, 69.25) mm, rotated rx 180 ry 0 rz -180 deg; joints [-146.402, -84.379, -25.361, 63.051, 38.373, -57.038]
  MoveL 4506 to (237.63, 158.7, 69.25) mm, rotated rx 180 ry 0 rz -180 deg; joints [-146.402, -84.379, -25.361, 63.051, 38.373, -57.038]
  Call Extruder(265.45104)
  MoveL 4507 to (237.3, 159.15, 69.25) mm, rotated rx 180 ry 0 rz 180 deg; joints [-146.352, -84.374, -25.371, 63.089, 38.417, -57.065]
  Call Extruder(266.27899)
  MoveL 4508 to (236.39, 160.19, 69.25) mm, rotated rx -180 ry 0 rz 180 deg; joints [-146.229, -84.335, -25.452, 63.151, 38.538, -57.09]
  Call Extruder(267.10694)
  MoveL 4509 to (235.35, 161.1, 69.25) mm, rotated rx 180 ry 0 rz 180 deg; joints [-146.109, -84.258, -25.607, 63.167, 38.675, -57.059]
  Call Extruder(267.27424)
  MoveL 4510 to (235.13, 161.27, 69.25) mm, rotated rx -180 ry 0 rz 180 deg; joints [-146.086, -84.238, -25.649, 63.164, 38.704, -57.044]
  MoveL 4511 to (235.13, 161.27, 69.25) mm, rotated rx -180 ry 0 rz 180 deg; joints [-146.086, -84.238, -25.649, 63.164, 38.704, -57.044]
  Call Extruder(267.60766)
  MoveL 4512 to (234.68, 161.59, 69.25) mm, rotated rx 180 ry 0 rz 180 deg; joints [-146.039, -84.197, -25.732, 63.157, 38.763, -57.016]
  MoveL 4513 to (234.68, 161.59, 69.25) mm, rotated rx 180 ry 0 rz 180 deg; joints [-146.039, -84.197, -25.732, 63.157, 38.763, -57.016]
  Call Extruder(267.93990)
  MoveL 4514 to (234.23, 161.92, 69.25) mm, rotated rx -180 ry 0 rz 180 deg; joints [-145.992, -84.156, -25.815, 63.151, 38.821, -56.987]
  MoveL 4515 to (234.23, 161.92, 69.25) mm, rotated rx -180 ry 0 rz 180 deg; joints [-145.992, -84.156, -25.815, 63.151, 38.821, -56.987]
  Call Extruder(268.05756)
  MoveL 4516 to (234.05, 162.02, 69.25) mm, rotated rx 180 ry 0 rz 180 deg; joints [-145.976, -84.138, -25.853, 63.144, 38.843, -56.971]
  MoveL 4517 to (234.05, 162.02, 69.25) mm, rotated rx 180 ry 0 rz 180 deg; joints [-145.976, -84.138, -25.853, 63.144, 38.843, -56.971]
  Call Extruder(268.26529)
  MoveL 4518 to (233.75, 162.2, 69.25) mm, rotated rx 180 ry 0 rz 180 deg; joints [-145.947, -84.105, -25.919, 63.131, 38.882, -56.942]
  MoveL 4519 to (233.75, 162.2, 69.25) mm, rotated rx 180 ry 0 rz 180 deg; joints [-145.947, -84.105, -25.919, 63.131, 38.882, -56.942]
  Call Extruder(268.47224)
  MoveL 4520 to (233.45, 162.37, 69.25) mm, rotated rx -180 ry 0 rz 180 deg; joints [-145.919, -84.072, -25.986, 63.118, 38.921, -56.913]
  MoveL 4521 to (233.45, 162.37, 69.25) mm, rotated rx -180 ry 0 rz 180 deg; joints [-145.919, -84.072, -25.986, 63.118, 38.921, -56.913]
  Call Extruder(268.67841)
  MoveL 4522 to (233.14, 162.55, 69.25) mm, rotated rx 180 ry 0 rz 180 deg; joints [-145.891, -84.04, -26.052, 63.105, 38.961, -56.884]
  MoveL 4523 to (233.14, 162.55, 69.25) mm, rotated rx 180 ry 0 rz 180 deg; joints [-145.891, -84.04, -26.052, 63.105, 38.961, -56.884]
  Call Extruder(268.86008)
  MoveL 4524 to (232.87, 162.69, 69.25) mm, rotated rx -180 ry 0 rz 180 deg; joints [-145.866, -84.008, -26.117, 63.09, 38.996, -56.854]
  MoveL 4525 to (232.87, 162.69, 69.25) mm, rotated rx -180 ry 0 rz 180 deg; joints [-145.866, -84.008, -26.117, 63.09, 38.996, -56.854]
  Call Extruder(269.01805)
  MoveL 4526 to (232.62, 162.8, 69.25) mm, rotated rx 180 ry 0 rz 180 deg; joints [-145.845, -83.977, -26.18, 63.073, 39.028, -56.822]
  MoveL 4527 to (232.62, 162.8, 69.25) mm, rotated rx 180 ry 0 rz 180 deg; joints [-145.845, -83.977, -26.18, 63.073, 39.028, -56.822]
  Call Extruder(269.17542)
  MoveL 4528 to (232.37, 162.9, 69.25) mm, rotated rx 180 ry 0 rz 180 deg; joints [-145.825, -83.946, -26.243, 63.056, 39.059, -56.791]
  MoveL 4529 to (232.37, 162.9, 69.25) mm, rotated rx 180 ry 0 rz 180 deg; joints [-145.825, -83.946, -26.243, 63.056, 39.059, -56.791]
  Call Extruder(269.35816)
  MoveL 4530 to (232.08, 163.03, 69.25) mm, rotated rx -180 ry 0 rz 180 deg; joints [-145.801, -83.91, -26.318, 63.034, 39.096, -56.753]
  MoveL 4531 to (232.08, 163.03, 69.25) mm, rotated rx -180 ry 0 rz 180 deg; joints [-145.801, -83.91, -26.318, 63.034, 39.096, -56.753]
  Call Extruder(269.54014)
  MoveL 4532 to (231.78, 163.15, 69.25) mm, rotated rx 180 ry 0 rz -180 deg; joints [-145.777, -83.873, -26.392, 63.013, 39.134, -56.715]
  MoveL 4533 to (231.78, 163.15, 69.25) mm, rotated rx 180 ry 0 rz -180 deg; joints [-145.777, -83.873, -26.392, 63.013, 39.134, -56.715]
  Call Extruder(269.68748)
  MoveL 4534 to (231.54, 163.24, 69.25) mm, rotated rx 180 ry 0 rz 180 deg; joints [-145.759, -83.842, -26.455, 62.995, 39.164, -56.683]
  MoveL 4535 to (231.54, 163.24, 69.25) mm, rotated rx 180 ry 0 rz 180 deg; joints [-145.759, -83.842, -26.455, 62.995, 39.164, -56.683]
  Call Extruder(269.80071)
  MoveL 4536 to (231.35, 163.3, 69.25) mm, rotated rx 180 ry 0 rz 180 deg; joints [-145.744, -83.817, -26.507, 62.978, 39.188, -56.655]
  MoveL 4537 to (231.35, 163.3, 69.25) mm, rotated rx 180 ry 0 rz 180 deg; joints [-145.744, -83.817, -26.507, 62.978, 39.188, -56.655]
  Call Extruder(269.91348)
  MoveL 4538 to (231.17, 163.36, 69.25) mm, rotated rx -180 ry 0 rz -180 deg; joints [-145.73, -83.792, -26.559, 62.962, 39.212, -56.627]
  MoveL 4539 to (231.17, 163.36, 69.25) mm, rotated rx -180 ry 0 rz -180 deg; joints [-145.73, -83.792, -26.559, 62.962, 39.212, -56.627]
  Call Extruder(270.02582)
  MoveL 4540 to (230.98, 163.42, 69.25) mm, rotated rx -180 ry 0 rz -180 deg; joints [-145.716, -83.766, -26.611, 62.945, 39.235, -56.599]
  MoveL 4541 to (230.98, 163.42, 69.25) mm, rotated rx -180 ry 0 rz -180 deg; joints [-145.716, -83.766, -26.611, 62.945, 39.235, -56.599]
  Call Extruder(270.13770)
  MoveL 4542 to (230.79, 163.48, 69.25) mm, rotated rx 180 ry 0 rz 180 deg; joints [-145.702, -83.741, -26.662, 62.928, 39.259, -56.572]
  MoveL 4543 to (230.79, 163.48, 69.25) mm, rotated rx 180 ry 0 rz 180 deg; joints [-145.702, -83.741, -26.662, 62.928, 39.259, -56.572]
  Call Extruder(270.25911)
  MoveL 4544 to (230.58, 163.55, 69.25) mm, rotated rx 180 ry 0 rz 180 deg; joints [-145.687, -83.713, -26.719, 62.91, 39.285, -56.541]
  MoveL 4545 to (230.58, 163.55, 69.25) mm, rotated rx 180 ry 0 rz 180 deg; joints [-145.687, -83.713, -26.719, 62.91, 39.285, -56.541]
  Call Extruder(270.38992)
  MoveL 4546 to (230.36, 163.62, 69.25) mm, rotated rx 180 ry 0 rz 180 deg; joints [-145.67, -83.683, -26.781, 62.89, 39.313, -56.508]
  MoveL 4547 to (230.36, 163.62, 69.25) mm, rotated rx 180 ry 0 rz 180 deg; joints [-145.67, -83.683, -26.781, 62.89, 39.313, -56.508]
  Call Extruder(270.52017)
  MoveL 4548 to (230.14, 163.68, 69.25) mm, rotated rx -180 ry 0 rz 180 deg; joints [-145.654, -83.652, -26.843, 62.87, 39.341, -56.474]
  MoveL 4549 to (230.14, 163.68, 69.25) mm, rotated rx -180 ry 0 rz 180 deg; joints [-145.654, -83.652, -26.843, 62.87, 39.341, -56.474]
  Call Extruder(270.64985)
  MoveL 4550 to (229.91, 163.75, 69.25) mm, rotated rx 180 ry 0 rz 180 deg; joints [-145.638, -83.622, -26.905, 62.85, 39.37, -56.441]
  MoveL 4551 to (229.91, 163.75, 69.25) mm, rotated rx 180 ry 0 rz 180 deg; joints [-145.638, -83.622, -26.905, 62.85, 39.37, -56.441]
  Call Extruder(270.77897)
  MoveL 4552 to (229.69, 163.82, 69.25) mm, rotated rx -180 ry 0 rz 180 deg; joints [-145.621, -83.591, -26.968, 62.83, 39.398, -56.407]
  MoveL 4553 to (229.69, 163.82, 69.25) mm, rotated rx -180 ry 0 rz 180 deg; joints [-145.621, -83.591, -26.968, 62.83, 39.398, -56.407]
  Call Extruder(270.89404)
  MoveL 4554 to (229.48, 163.86, 69.25) mm, rotated rx 180 ry 0 rz 180 deg; joints [-145.607, -83.562, -27.028, 62.808, 39.423, -56.373]
  MoveL 4555 to (229.48, 163.86, 69.25) mm, rotated rx 180 ry 0 rz 180 deg; joints [-145.607, -83.562, -27.028, 62.808, 39.423, -56.373]
  Call Extruder(271.00867)
  MoveL 4556 to (229.28, 163.91, 69.25) mm, rotated rx 180 ry 0 rz -180 deg; joints [-145.594, -83.532, -27.088, 62.787, 39.449, -56.34]
  MoveL 4557 to (229.28, 163.91, 69.25) mm, rotated rx 180 ry 0 rz -180 deg; joints [-145.594, -83.532, -27.088, 62.787, 39.449, -56.34]
  Call Extruder(271.12284)
  MoveL 4558 to (229.08, 163.95, 69.25) mm, rotated rx -180 ry 0 rz -180 deg; joints [-145.58, -83.503, -27.148, 62.766, 39.474, -56.306]
  MoveL 4559 to (229.08, 163.95, 69.25) mm, rotated rx -180 ry 0 rz -180 deg; joints [-145.58, -83.503, -27.148, 62.766, 39.474, -56.306]
  Call Extruder(271.23656)
  MoveL 4560 to (228.87, 164, 69.25) mm, rotated rx -180 ry 0 rz 180 deg; joints [-145.566, -83.473, -27.209, 62.744, 39.5, -56.272]
  MoveL 4561 to (228.87, 164, 69.25) mm, rotated rx -180 ry 0 rz 180 deg; joints [-145.566, -83.473, -27.209, 62.744, 39.5, -56.272]
  Call Extruder(271.36198)
  MoveL 4562 to (228.65, 164.04, 69.25) mm, rotated rx 180 ry 0 rz 180 deg; joints [-145.551, -83.44, -27.276, 62.72, 39.528, -56.234]
  MoveL 4563 to (228.65, 164.04, 69.25) mm, rotated rx 180 ry 0 rz 180 deg; joints [-145.551, -83.44, -27.276, 62.72, 39.528, -56.234]
  Call Extruder(271.49895)
  MoveL 4564 to (228.4, 164.09, 69.25) mm, rotated rx 180 ry 0 rz 180 deg; joints [-145.535, -83.404, -27.35, 62.694, 39.559, -56.192]
  MoveL 4565 to (228.4, 164.09, 69.25) mm, rotated rx 180 ry 0 rz 180 deg; joints [-145.535, -83.404, -27.35, 62.694, 39.559, -56.192]
  Call Extruder(271.63532)
  MoveL 4566 to (228.15, 164.14, 69.25) mm, rotated rx 180 ry 0 rz 180 deg; joints [-145.518, -83.368, -27.425, 62.667, 39.59, -56.15]
  MoveL 4567 to (228.15, 164.14, 69.25) mm, rotated rx 180 ry 0 rz 180 deg; joints [-145.518, -83.368, -27.425, 62.667, 39.59, -56.15]
  Call Extruder(271.77108)
  MoveL 4568 to (227.9, 164.19, 69.25) mm, rotated rx -180 ry 0 rz 180 deg; joints [-145.502, -83.332, -27.499, 62.641, 39.621, -56.109]
  MoveL 4569 to (227.9, 164.19, 69.25) mm, rotated rx -180 ry 0 rz 180 deg; joints [-145.502, -83.332, -27.499, 62.641, 39.621, -56.109]
  Call Extruder(271.90623)
  MoveL 4570 to (227.65, 164.24, 69.25) mm, rotated rx -180 ry 0 rz 180 deg; joints [-145.485, -83.296, -27.573, 62.615, 39.652, -56.067]
  MoveL 4571 to (227.65, 164.24, 69.25) mm, rotated rx -180 ry 0 rz 180 deg; joints [-145.485, -83.296, -27.573, 62.615, 39.652, -56.067]
  Call Extruder(272.04076)
  MoveL 4572 to (227.4, 164.29, 69.25) mm, rotated rx -180 ry 0 rz 180 deg; joints [-145.469, -83.26, -27.646, 62.589, 39.683, -56.026]
  MoveL 4573 to (227.4, 164.29, 69.25) mm, rotated rx -180 ry 0 rz 180 deg; joints [-145.469, -83.26, -27.646, 62.589, 39.683, -56.026]
  Call Extruder(272.17469)
  MoveL 4574 to (227.15, 164.34, 69.25) mm, rotated rx 180 ry 0 rz 180 deg; joints [-145.453, -83.224, -27.72, 62.563, 39.714, -55.984]
  MoveL 4575 to (227.15, 164.34, 69.25) mm, rotated rx 180 ry 0 rz 180 deg; joints [-145.453, -83.224, -27.72, 62.563, 39.714, -55.984]
  Call Extruder(272.32256)
  MoveL 4576 to (226.87, 164.39, 69.25) mm, rotated rx 180 ry 0 rz -180 deg; joints [-145.435, -83.183, -27.803, 62.534, 39.749, -55.938]
  MoveL 4577 to (226.87, 164.39, 69.25) mm, rotated rx 180 ry 0 rz -180 deg; joints [-145.435, -83.183, -27.803, 62.534, 39.749, -55.938]
  Call Extruder(272.48429)
  MoveL 4578 to (226.57, 164.44, 69.25) mm, rotated rx 180 ry 0 rz 180 deg; joints [-145.415, -83.138, -27.895, 62.5, 39.787, -55.885]
  MoveL 4579 to (226.57, 164.44, 69.25) mm, rotated rx 180 ry 0 rz 180 deg; joints [-145.415, -83.138, -27.895, 62.5, 39.787, -55.885]
  Call Extruder(272.64531)
  MoveL 4580 to (226.26, 164.49, 69.25) mm, rotated rx -180 ry 0 rz 180 deg; joints [-145.396, -83.093, -27.988, 62.466, 39.824, -55.832]
  MoveL 4581 to (226.26, 164.49, 69.25) mm, rotated rx -180 ry 0 rz 180 deg; joints [-145.396, -83.093, -27.988, 62.466, 39.824, -55.832]
  Call Extruder(272.80559)
  MoveL 4582 to (225.95, 164.53, 69.25) mm, rotated rx 180 ry 0 rz 180 deg; joints [-145.377, -83.047, -28.08, 62.433, 39.862, -55.78]
  MoveL 4583 to (225.95, 164.53, 69.25) mm, rotated rx 180 ry 0 rz 180 deg; joints [-145.377, -83.047, -28.08, 62.433, 39.862, -55.78]
  Call Extruder(272.96514)
  MoveL 4584 to (225.65, 164.58, 69.25) mm, rotated rx -180 ry 0 rz 180 deg; joints [-145.357, -83.003, -28.172, 62.4, 39.9, -55.728]
  MoveL 4585 to (225.65, 164.58, 69.25) mm, rotated rx -180 ry 0 rz 180 deg; joints [-145.357, -83.003, -28.172, 62.4, 39.9, -55.728]
  Call Extruder(273.12397)
  MoveL 4586 to (225.34, 164.63, 69.25) mm, rotated rx -180 ry 0 rz 180 deg; joints [-145.338, -82.958, -28.264, 62.368, 39.938, -55.676]
  MoveL 4587 to (225.34, 164.63, 69.25) mm, rotated rx -180 ry 0 rz 180 deg; joints [-145.338, -82.958, -28.264, 62.368, 39.938, -55.676]
  Call Extruder(273.30264)
  MoveL 4588 to (225, 164.68, 69.25) mm, rotated rx 180 ry 0 rz 180 deg; joints [-145.317, -82.906, -28.37, 62.329, 39.981, -55.615]
  MoveL 4589 to (225, 164.68, 69.25) mm, rotated rx 180 ry 0 rz 180 deg; joints [-145.317, -82.906, -28.37, 62.329, 39.981, -55.615]
  Call Extruder(273.50108)
  MoveL 4590 to (224.61, 164.72, 69.25) mm, rotated rx 180 ry 0 rz -180 deg; joints [-145.293, -82.848, -28.489, 62.285, 40.028, -55.547]
  MoveL 4591 to (224.61, 164.72, 69.25) mm, rotated rx 180 ry 0 rz -180 deg; joints [-145.293, -82.848, -28.489, 62.285, 40.028, -55.547]
  Call Extruder(273.69866)
  MoveL 4592 to (224.22, 164.77, 69.25) mm, rotated rx -180 ry 0 rz 180 deg; joints [-145.27, -82.79, -28.608, 62.242, 40.076, -55.479]
  MoveL 4593 to (224.22, 164.77, 69.25) mm, rotated rx -180 ry 0 rz 180 deg; joints [-145.27, -82.79, -28.608, 62.242, 40.076, -55.479]
  Call Extruder(273.89536)
  MoveL 4594 to (223.83, 164.82, 69.25) mm, rotated rx 180 ry 0 rz 180 deg; joints [-145.246, -82.732, -28.727, 62.198, 40.124, -55.411]
  MoveL 4595 to (223.83, 164.82, 69.25) mm, rotated rx 180 ry 0 rz 180 deg; joints [-145.246, -82.732, -28.727, 62.198, 40.124, -55.411]
  Call Extruder(274.09120)
  MoveL 4596 to (223.45, 164.86, 69.25) mm, rotated rx -180 ry 0 rz 180 deg; joints [-145.223, -82.675, -28.845, 62.155, 40.171, -55.344]
  MoveL 4597 to (223.45, 164.86, 69.25) mm, rotated rx -180 ry 0 rz 180 deg; joints [-145.223, -82.675, -28.845, 62.155, 40.171, -55.344]
  Call Extruder(274.38656)
  MoveL 4598 to (222.86, 164.91, 69.25) mm, rotated rx -180 ry 0 rz 180 deg; joints [-145.189, -82.585, -29.029, 62.087, 40.244, -55.237]
  MoveL 4599 to (222.86, 164.91, 69.25) mm, rotated rx -180 ry 0 rz 180 deg; joints [-145.189, -82.585, -29.029, 62.087, 40.244, -55.237]
  Call Extruder(274.68059)
  MoveL 4600 to (222.27, 164.96, 69.25) mm, rotated rx -180 ry 0 rz 180 deg; joints [-145.155, -82.496, -29.213, 62.018, 40.316, -55.132]
  MoveL 4601 to (222.27, 164.96, 69.25) mm, rotated rx -180 ry 0 rz 180 deg; joints [-145.155, -82.496, -29.213, 62.018, 40.316, -55.132]
  Call Extruder(274.97329)
  MoveL 4602 to (221.68, 165, 69.25) mm, rotated rx -180 ry 0 rz -180 deg; joints [-145.121, -82.407, -29.395, 61.951, 40.388, -55.027]
  MoveL 4603 to (221.68, 165, 69.25) mm, rotated rx -180 ry 0 rz -180 deg; joints [-145.121, -82.407, -29.395, 61.951, 40.388, -55.027]
  Call Extruder(275.54673)
  MoveL 4604 to (220.52, 165.05, 69.25) mm, rotated rx 180 ry 0 rz 180 deg; joints [-145.056, -82.228, -29.764, 61.812, 40.529, -54.813]
  MoveL 4605 to (220.52, 165.05, 69.25) mm, rotated rx 180 ry 0 rz 180 deg; joints [-145.056, -82.228, -29.764, 61.812, 40.529, -54.813]
  Call Extruder(276.26074)
  MoveL 4606 to (219.06, 165.09, 69.25) mm, rotated rx -180 ry 0 rz -180 deg; joints [-144.977, -82.004, -30.224, 61.64, 40.706, -54.546]
  Call Extruder(393.10748)
  MoveL 4607 to (-19.06, 165.09, 69.25) mm, rotated rx 180 ry 0 rz 180 deg; joints [-127.434, -61.598, -75.892, 60.564, 65.749, -36.05]
  Call Extruder(393.53608)
  MoveL 4608 to (-19.94, 165.07, 69.25) mm, rotated rx -180 ry 0 rz -180 deg; joints [-127.348, -61.555, -76.001, 60.614, 65.832, -36.018]
  MoveL 4609 to (-19.94, 165.07, 69.25) mm, rotated rx -180 ry 0 rz -180 deg; joints [-127.348, -61.555, -76.001, 60.614, 65.832, -36.018]
  Call Extruder(394.10954)
  MoveL 4610 to (-21.1, 165.03, 69.25) mm, rotated rx 180 ry 0 rz 180 deg; joints [-127.235, -61.498, -76.148, 60.68, 65.943, -35.973]
  MoveL 4611 to (-21.1, 165.03, 69.25) mm, rotated rx 180 ry 0 rz 180 deg; joints [-127.235, -61.498, -76.148, 60.68, 65.943, -35.973]
  Call Extruder(394.54383)
  MoveL 4612 to (-21.97, 164.98, 69.25) mm, rotated rx 180 ry 0 rz -180 deg; joints [-127.15, -61.453, -76.261, 60.729, 66.026, -35.938]
  MoveL 4613 to (-21.97, 164.98, 69.25) mm, rotated rx 180 ry 0 rz -180 deg; joints [-127.15, -61.453, -76.261, 60.729, 66.026, -35.938]
  Call Extruder(394.83786)
  MoveL 4614 to (-22.56, 164.93, 69.25) mm, rotated rx -180 ry 0 rz 180 deg; joints [-127.093, -61.423, -76.34, 60.76, 66.083, -35.913]
  MoveL 4615 to (-22.56, 164.93, 69.25) mm, rotated rx -180 ry 0 rz 180 deg; joints [-127.093, -61.423, -76.34, 60.76, 66.083, -35.913]
  Call Extruder(395.13322)
  MoveL 4616 to (-23.15, 164.89, 69.25) mm, rotated rx -180 ry 0 rz 180 deg; joints [-127.037, -61.392, -76.418, 60.791, 66.139, -35.888]
  MoveL 4617 to (-23.15, 164.89, 69.25) mm, rotated rx -180 ry 0 rz 180 deg; joints [-127.037, -61.392, -76.418, 60.791, 66.139, -35.888]
  Call Extruder(395.37944)
  MoveL 4618 to (-23.64, 164.84, 69.25) mm, rotated rx 180 ry 0 rz 180 deg; joints [-126.991, -61.367, -76.483, 60.817, 66.185, -35.866]
  MoveL 4619 to (-23.64, 164.84, 69.25) mm, rotated rx 180 ry 0 rz 180 deg; joints [-126.991, -61.367, -76.483, 60.817, 66.185, -35.866]
  Call Extruder(395.57615)
  MoveL 4620 to (-24.03, 164.79, 69.25) mm, rotated rx 180 ry 0 rz -180 deg; joints [-126.955, -61.346, -76.537, 60.836, 66.222, -35.847]
  MoveL 4621 to (-24.03, 164.79, 69.25) mm, rotated rx 180 ry 0 rz -180 deg; joints [-126.955, -61.346, -76.537, 60.836, 66.222, -35.847]
  Call Extruder(395.77372)
  MoveL 4622 to (-24.42, 164.75, 69.25) mm, rotated rx 180 ry 0 rz 180 deg; joints [-126.919, -61.325, -76.591, 60.855, 66.259, -35.829]
  MoveL 4623 to (-24.42, 164.75, 69.25) mm, rotated rx 180 ry 0 rz 180 deg; joints [-126.919, -61.325, -76.591, 60.855, 66.259, -35.829]
  Call Extruder(395.97216)
  MoveL 4624 to (-24.8, 164.7, 69.25) mm, rotated rx 180 ry 0 rz 180 deg; joints [-126.883, -61.304, -76.644, 60.874, 66.296, -35.811]
  MoveL 4625 to (-24.8, 164.7, 69.25) mm, rotated rx 180 ry 0 rz 180 deg; joints [-126.883, -61.304, -76.644, 60.874, 66.296, -35.811]
  Call Extruder(396.17147)
  MoveL 4626 to (-25.19, 164.66, 69.25) mm, rotated rx -180 ry 0 rz 180 deg; joints [-126.847, -61.283, -76.698, 60.894, 66.333, -35.792]
  MoveL 4627 to (-25.19, 164.66, 69.25) mm, rotated rx -180 ry 0 rz 180 deg; joints [-126.847, -61.283, -76.698, 60.894, 66.333, -35.792]
  Call Extruder(396.33030)
  MoveL 4628 to (-25.5, 164.61, 69.25) mm, rotated rx 180 ry 0 rz 180 deg; joints [-126.82, -61.266, -76.742, 60.908, 66.362, -35.777]
  MoveL 4629 to (-25.5, 164.61, 69.25) mm, rotated rx 180 ry 0 rz 180 deg; joints [-126.82, -61.266, -76.742, 60.908, 66.362, -35.777]
  Call Extruder(396.48986)
  MoveL 4630 to (-25.8, 164.56, 69.25) mm, rotated rx -180 ry 0 rz 180 deg; joints [-126.792, -61.249, -76.786, 60.922, 66.391, -35.761]
  MoveL 4631 to (-25.8, 164.56, 69.25) mm, rotated rx -180 ry 0 rz 180 deg; joints [-126.792, -61.249, -76.786, 60.922, 66.391, -35.761]
  Call Extruder(396.65015)
  MoveL 4632 to (-26.11, 164.51, 69.25) mm, rotated rx 180 ry 0 rz 180 deg; joints [-126.765, -61.232, -76.83, 60.936, 66.421, -35.745]
  MoveL 4633 to (-26.11, 164.51, 69.25) mm, rotated rx 180 ry 0 rz 180 deg; joints [-126.765, -61.232, -76.83, 60.936, 66.421, -35.745]
  Call Extruder(396.81116)
  MoveL 4634 to (-26.41, 164.46, 69.25) mm, rotated rx 180 ry 0 rz 180 deg; joints [-126.737, -61.215, -76.874, 60.95, 66.45, -35.729]
  MoveL 4635 to (-26.41, 164.46, 69.25) mm, rotated rx 180 ry 0 rz 180 deg; joints [-126.737, -61.215, -76.874, 60.95, 66.45, -35.729]
  Call Extruder(396.97291)
  MoveL 4636 to (-26.72, 164.41, 69.25) mm, rotated rx 180 ry 0 rz 180 deg; joints [-126.71, -61.198, -76.917, 60.965, 66.479, -35.713]
  MoveL 4637 to (-26.72, 164.41, 69.25) mm, rotated rx 180 ry 0 rz 180 deg; joints [-126.71, -61.198, -76.917, 60.965, 66.479, -35.713]
  Call Extruder(397.13538)
  MoveL 4638 to (-27.03, 164.36, 69.25) mm, rotated rx -180 ry 0 rz 180 deg; joints [-126.682, -61.181, -76.961, 60.979, 66.508, -35.697]
  MoveL 4639 to (-27.03, 164.36, 69.25) mm, rotated rx -180 ry 0 rz 180 deg; joints [-126.682, -61.181, -76.961, 60.979, 66.508, -35.697]
  Call Extruder(397.26930)
  MoveL 4640 to (-27.27, 164.32, 69.25) mm, rotated rx 180 ry 0 rz 180 deg; joints [-126.66, -61.166, -76.999, 60.989, 66.532, -35.683]
  MoveL 4641 to (-27.27, 164.32, 69.25) mm, rotated rx 180 ry 0 rz 180 deg; joints [-126.66, -61.166, -76.999, 60.989, 66.532, -35.683]
  Call Extruder(397.40384)
  MoveL 4642 to (-27.52, 164.27, 69.25) mm, rotated rx -180 ry 0 rz 180 deg; joints [-126.638, -61.152, -77.036, 61, 66.556, -35.669]
  MoveL 4643 to (-27.52, 164.27, 69.25) mm, rotated rx -180 ry 0 rz 180 deg; joints [-126.638, -61.152, -77.036, 61, 66.556, -35.669]
  Call Extruder(397.53899)
  MoveL 4644 to (-27.77, 164.22, 69.25) mm, rotated rx 180 ry 0 rz 180 deg; joints [-126.617, -61.137, -77.073, 61.011, 66.579, -35.655]
  MoveL 4645 to (-27.77, 164.22, 69.25) mm, rotated rx 180 ry 0 rz 180 deg; joints [-126.617, -61.137, -77.073, 61.011, 66.579, -35.655]
  Call Extruder(397.67474)
  MoveL 4646 to (-28.02, 164.17, 69.25) mm, rotated rx 180 ry 0 rz 180 deg; joints [-126.595, -61.123, -77.11, 61.021, 66.603, -35.641]
  MoveL 4647 to (-28.02, 164.17, 69.25) mm, rotated rx 180 ry 0 rz 180 deg; joints [-126.595, -61.123, -77.11, 61.021, 66.603, -35.641]
  Call Extruder(397.81111)
  MoveL 4648 to (-28.27, 164.12, 69.25) mm, rotated rx -180 ry 0 rz 180 deg; joints [-126.573, -61.108, -77.148, 61.032, 66.627, -35.627]
  MoveL 4649 to (-28.27, 164.12, 69.25) mm, rotated rx -180 ry 0 rz 180 deg; joints [-126.573, -61.108, -77.148, 61.032, 66.627, -35.627]
  Call Extruder(397.89597)
  MoveL 4650 to (-28.42, 164.09, 69.25) mm, rotated rx 180 ry 0 rz -180 deg; joints [-126.559, -61.099, -77.171, 61.039, 66.642, -35.619]
  Set speed (130.0 mm/s)
  MoveL 4651 to (-31.76, 163.31, 69.25) mm, rotated rx 180 ry 0 rz 180 deg; joints [-126.274, -60.901, -77.684, 61.173, 66.959, -35.418]
  MoveL 4652 to (-31.76, 163.31, 78.65) mm, rotated rx 180 ry 0 rz 180 deg; joints [-126.274, -59.612, -78.328, 61.416, 66.65, -36.033]
  Call Extruder(395.89597)
  Set speed (40.0 mm/s)
  MoveL 4653 to (-31.76, 163.31, 78.65) mm, rotated rx 180 ry 0 rz 180 deg; joints [-126.274, -59.612, -78.328, 61.416, 66.65, -36.033]
  Call Extruder(0.00000)
  Set speed (130.0 mm/s)
  MoveL 4654 to (-31.64, 163.21, 78.65) mm, rotated rx 180 ry 0 rz -180 deg; joints [-126.294, -59.611, -78.33, 61.397, 66.638, -36.025]
  Call Extruder(2.00000)
  Set speed (40.0 mm/s)
  MoveL 4655 to (-31.64, 163.21, 78.65) mm, rotated rx 180 ry 0 rz -180 deg; joints [-126.294, -59.611, -78.33, 61.397, 66.638, -36.025]
  Set speed (30.0 mm/s)
  MoveL 4656 to (-31.64, 163.21, 78.65) mm, rotated rx 180 ry 0 rz -180 deg; joints [-126.294, -59.611, -78.33, 61.397, 66.638, -36.025]
  Call Extruder(2.18198)
  MoveL 4657 to (-31.93, 163.09, 78.65) mm, rotated rx 180 ry 0 rz -180 deg; joints [-126.273, -59.59, -78.383, 61.404, 66.666, -36.002]
